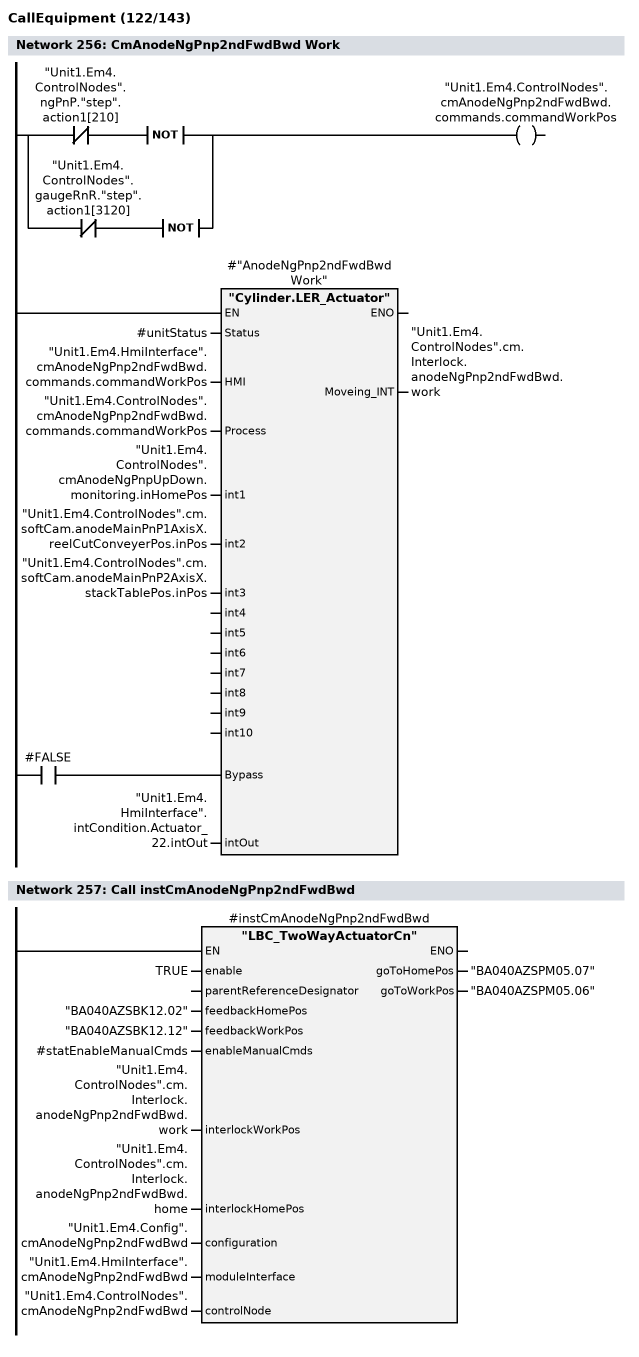
   RUNG wire#powerrail
      I_Contact( "Unit1.Em4.ControlNodes".ngPnP."step".action1[210] )
      Not()
      wire#w1
      Coil( "Unit1.Em4.ControlNodes".cmAnodeNgPnp2ndFwdBwd.commands.commandWorkPos )
   END_RUNG
   RUNG wire#powerrail
      I_Contact( "Unit1.Em4.ControlNodes".gaugeRnR."step".action1[3120] )
      Not()
   END_RUNG wire#w1
   RUNG wire#powerrail
      #"AnodeNgPnp2ndFwdBwd Work"(Bypass := wire#w2, Status := #unitStatus, HMI := "Unit1.Em4.HmiInterface".cmAnodeNgPnp2ndFwdBwd.commands.commandWorkPos, Process := "Unit1.Em4.ControlNodes".cmAnodeNgPnp2ndFwdBwd.commands.commandWorkPos, int1 := "Unit1.Em4.ControlNodes".cmAnodeNgPnpUpDown.monitoring.inHomePos, int2 := "Unit1.Em4.ControlNodes".cm.softCam.anodeMainPnP1AxisX.reelCutConveyerPos.inPos, int3 := "Unit1.Em4.ControlNodes".cm.softCam.anodeMainPnP2AxisX.stackTablePos.inPos, int4 :=, int5 :=, int6 :=, int7 :=, int8 :=, int9 :=, int10 :=, intOut := "Unit1.Em4.HmiInterface".intCondition.Actuator_22.intOut, Moveing_INT => "Unit1.Em4.ControlNodes".cm.Interlock.anodeNgPnp2ndFwdBwd.work)
   END_RUNG
   RUNG wire#powerrail
      Contact( #FALSE )
   END_RUNG wire#w2
   // the same network as SCL:
   "Unit1.Em4.ControlNodes".cmAnodeNgPnp2ndFwdBwd.commands.commandWorkPos := NOT (NOT "Unit1.Em4.ControlNodes".ngPnP."step".action1[210]) OR NOT (NOT "Unit1.Em4.ControlNodes".gaugeRnR."step".action1[3120]);
   #"AnodeNgPnp2ndFwdBwd Work"(Status := #unitStatus,   // "Cylinder.LER_Actuator"
                           HMI := "Unit1.Em4.HmiInterface".cmAnodeNgPnp2ndFwdBwd.commands.commandWorkPos,
                           Process := "Unit1.Em4.ControlNodes".cmAnodeNgPnp2ndFwdBwd.commands.commandWorkPos,
                           int1 := "Unit1.Em4.ControlNodes".cmAnodeNgPnpUpDown.monitoring.inHomePos,
                           int2 := "Unit1.Em4.ControlNodes".cm.softCam.anodeMainPnP1AxisX.reelCutConveyerPos.inPos,
                           int3 := "Unit1.Em4.ControlNodes".cm.softCam.anodeMainPnP2AxisX.stackTablePos.inPos,
                           Bypass := #FALSE,
                           intOut := "Unit1.Em4.HmiInterface".intCondition.Actuator_22.intOut,
                           Moveing_INT => "Unit1.Em4.ControlNodes".cm.Interlock.anodeNgPnp2ndFwdBwd.work);
END_REGION

REGION Network 257: Call instCmAnodeNgPnp2ndFwdBwd
   RUNG wire#powerrail
      #instCmAnodeNgPnp2ndFwdBwd(enable := TRUE, parentReferenceDesignator :=, feedbackHomePos := "BA040AZSBK12.02", feedbackWorkPos := "BA040AZSBK12.12", enableManualCmds := #statEnableManualCmds, interlockWorkPos := "Unit1.Em4.ControlNodes".cm.Interlock.anodeNgPnp2ndFwdBwd.work, interlockHomePos := "Unit1.Em4.ControlNodes".cm.Interlock.anodeNgPnp2ndFwdBwd.home, configuration := "Unit1.Em4.Config".cmAnodeNgPnp2ndFwdBwd, moduleInterface := "Unit1.Em4.HmiInterface".cmAnodeNgPnp2ndFwdBwd, controlNode := "Unit1.Em4.ControlNodes".cmAnodeNgPnp2ndFwdBwd, goToHomePos => "BA040AZSPM05.07", goToWorkPos => "BA040AZSPM05.06")
   END_RUNG
   // the same network as SCL:
   #instCmAnodeNgPnp2ndFwdBwd(enable := TRUE,   // "LBC_TwoWayActuatorCn"
                           feedbackHomePos := "BA040AZSBK12.02",
                           feedbackWorkPos := "BA040AZSBK12.12",
                           enableManualCmds := #statEnableManualCmds,
                           interlockWorkPos := "Unit1.Em4.ControlNodes".cm.Interlock.anodeNgPnp2ndFwdBwd.work,
                           interlockHomePos := "Unit1.Em4.ControlNodes".cm.Interlock.anodeNgPnp2ndFwdBwd.home,
                           configuration := "Unit1.Em4.Config".cmAnodeNgPnp2ndFwdBwd,
                           moduleInterface := "Unit1.Em4.HmiInterface".cmAnodeNgPnp2ndFwdBwd,
                           controlNode := "Unit1.Em4.ControlNodes".cmAnodeNgPnp2ndFwdBwd,
                           goToHomePos => "BA040AZSPM05.07",
                           goToWorkPos => "BA040AZSPM05.06");
END_REGION

REGION Network 259: CmAnodeMaintenanceMovingFixFrontRearFwdBwd Home
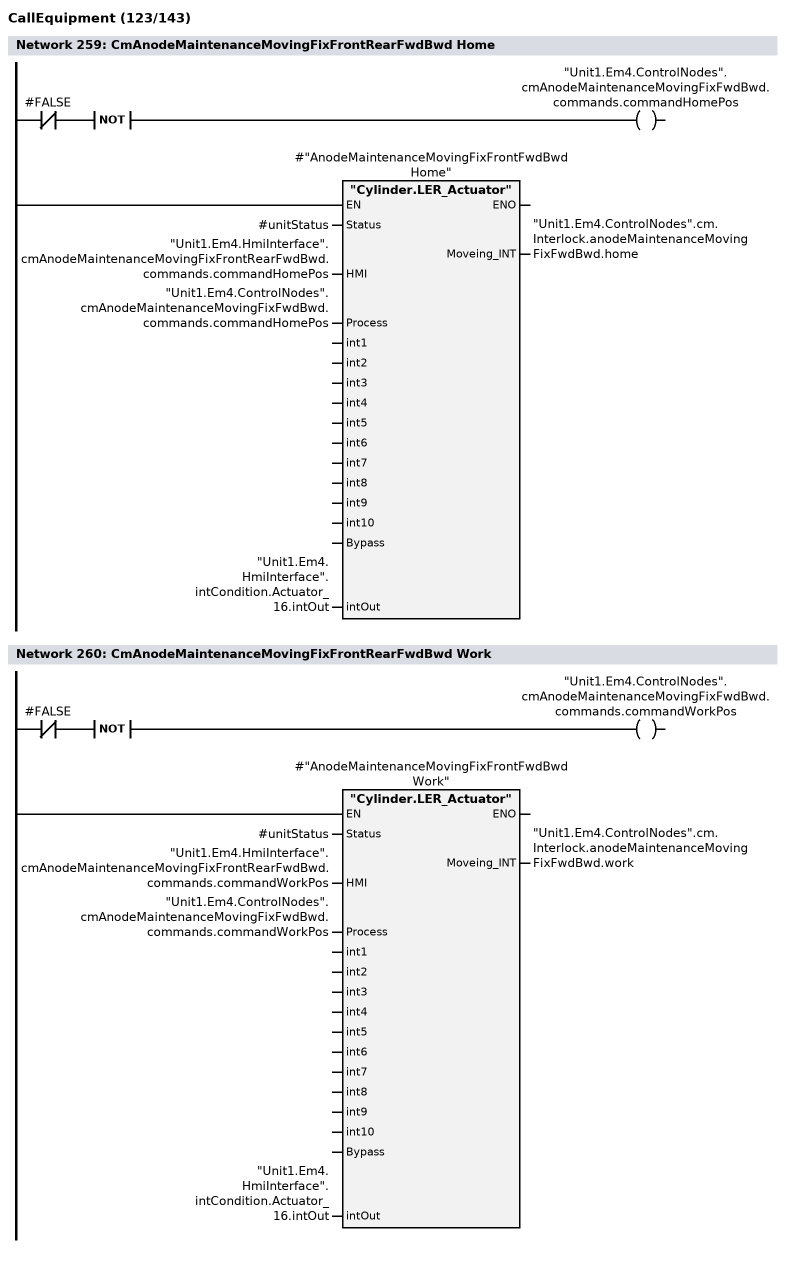
   RUNG wire#powerrail
      I_Contact( #FALSE )
      Not()
      Coil( "Unit1.Em4.ControlNodes".cmAnodeMaintenanceMovingFixFwdBwd.commands.commandHomePos )
   END_RUNG
   RUNG wire#powerrail
      #"AnodeMaintenanceMovingFixFrontFwdBwd Home"(Status := #unitStatus, HMI := "Unit1.Em4.HmiInterface".cmAnodeMaintenanceMovingFixFrontRearFwdBwd.commands.commandHomePos, Process := "Unit1.Em4.ControlNodes".cmAnodeMaintenanceMovingFixFwdBwd.commands.commandHomePos, int1 :=, int2 :=, int3 :=, int4 :=, int5 :=, int6 :=, int7 :=, int8 :=, int9 :=, int10 :=, Bypass :=, intOut := "Unit1.Em4.HmiInterface".intCondition.Actuator_16.intOut, Moveing_INT => "Unit1.Em4.ControlNodes".cm.Interlock.anodeMaintenanceMovingFixFwdBwd.home)
   END_RUNG
   // the same network as SCL:
   "Unit1.Em4.ControlNodes".cmAnodeMaintenanceMovingFixFwdBwd.commands.commandHomePos := NOT (NOT #FALSE);
   #"AnodeMaintenanceMovingFixFrontFwdBwd Home"(Status := #unitStatus,   // "Cylinder.LER_Actuator"
                           HMI := "Unit1.Em4.HmiInterface".cmAnodeMaintenanceMovingFixFrontRearFwdBwd.commands.commandHomePos,
                           Process := "Unit1.Em4.ControlNodes".cmAnodeMaintenanceMovingFixFwdBwd.commands.commandHomePos,
                           intOut := "Unit1.Em4.HmiInterface".intCondition.Actuator_16.intOut,
                           Moveing_INT => "Unit1.Em4.ControlNodes".cm.Interlock.anodeMaintenanceMovingFixFwdBwd.home);
END_REGION

REGION Network 260: CmAnodeMaintenanceMovingFixFrontRearFwdBwd Work
   RUNG wire#powerrail
      I_Contact( #FALSE )
      Not()
      Coil( "Unit1.Em4.ControlNodes".cmAnodeMaintenanceMovingFixFwdBwd.commands.commandWorkPos )
   END_RUNG
   RUNG wire#powerrail
      #"AnodeMaintenanceMovingFixFrontFwdBwd Work"(Status := #unitStatus, HMI := "Unit1.Em4.HmiInterface".cmAnodeMaintenanceMovingFixFrontRearFwdBwd.commands.commandWorkPos, Process := "Unit1.Em4.ControlNodes".cmAnodeMaintenanceMovingFixFwdBwd.commands.commandWorkPos, int1 :=, int2 :=, int3 :=, int4 :=, int5 :=, int6 :=, int7 :=, int8 :=, int9 :=, int10 :=, Bypass :=, intOut := "Unit1.Em4.HmiInterface".intCondition.Actuator_16.intOut, Moveing_INT => "Unit1.Em4.ControlNodes".cm.Interlock.anodeMaintenanceMovingFixFwdBwd.work)
   END_RUNG
   // the same network as SCL:
   "Unit1.Em4.ControlNodes".cmAnodeMaintenanceMovingFixFwdBwd.commands.commandWorkPos := NOT (NOT #FALSE);
   #"AnodeMaintenanceMovingFixFrontFwdBwd Work"(Status := #unitStatus,   // "Cylinder.LER_Actuator"
                           HMI := "Unit1.Em4.HmiInterface".cmAnodeMaintenanceMovingFixFrontRearFwdBwd.commands.commandWorkPos,
                           Process := "Unit1.Em4.ControlNodes".cmAnodeMaintenanceMovingFixFwdBwd.commands.commandWorkPos,
                           intOut := "Unit1.Em4.HmiInterface".intCondition.Actuator_16.intOut,
                           Moveing_INT => "Unit1.Em4.ControlNodes".cm.Interlock.anodeMaintenanceMovingFixFwdBwd.work);
END_REGION

REGION Network 261: Call instCmAnodeMaintenanceMovingFixFrontRearFwdBwd
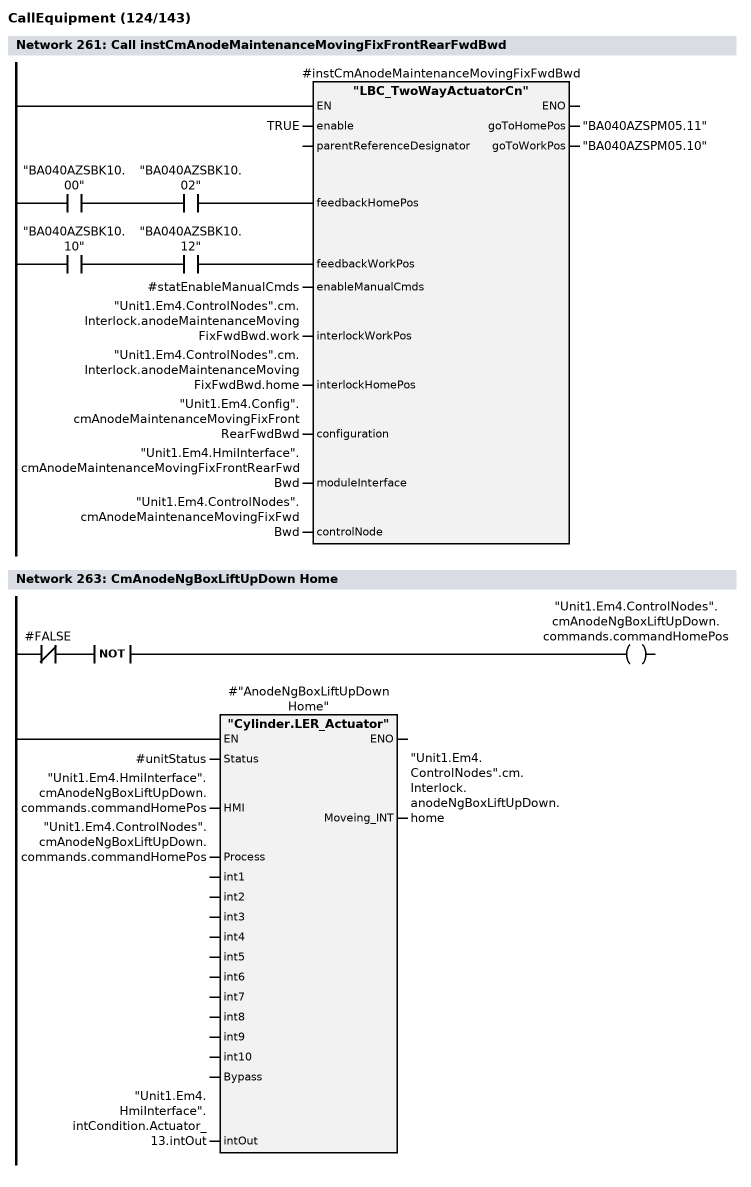
   RUNG wire#powerrail
      #instCmAnodeMaintenanceMovingFixFwdBwd(feedbackHomePos := wire#w1, feedbackWorkPos := wire#w2, enable := TRUE, parentReferenceDesignator :=, enableManualCmds := #statEnableManualCmds, interlockWorkPos := "Unit1.Em4.ControlNodes".cm.Interlock.anodeMaintenanceMovingFixFwdBwd.work, interlockHomePos := "Unit1.Em4.ControlNodes".cm.Interlock.anodeMaintenanceMovingFixFwdBwd.home, configuration := "Unit1.Em4.Config".cmAnodeMaintenanceMovingFixFrontRearFwdBwd, moduleInterface := "Unit1.Em4.HmiInterface".cmAnodeMaintenanceMovingFixFrontRearFwdBwd, controlNode := "Unit1.Em4.ControlNodes".cmAnodeMaintenanceMovingFixFwdBwd, goToHomePos => "BA040AZSPM05.11", goToWorkPos => "BA040AZSPM05.10")
   END_RUNG
   RUNG wire#powerrail
      Contact( "BA040AZSBK10.00" )
      Contact( "BA040AZSBK10.02" )
   END_RUNG wire#w1
   RUNG wire#powerrail
      Contact( "BA040AZSBK10.10" )
      Contact( "BA040AZSBK10.12" )
   END_RUNG wire#w2
   // the same network as SCL:
   #instCmAnodeMaintenanceMovingFixFwdBwd(enable := TRUE,   // "LBC_TwoWayActuatorCn"
                           feedbackHomePos := "BA040AZSBK10.00" AND "BA040AZSBK10.02",
                           feedbackWorkPos := "BA040AZSBK10.10" AND "BA040AZSBK10.12",
                           enableManualCmds := #statEnableManualCmds,
                           interlockWorkPos := "Unit1.Em4.ControlNodes".cm.Interlock.anodeMaintenanceMovingFixFwdBwd.work,
                           interlockHomePos := "Unit1.Em4.ControlNodes".cm.Interlock.anodeMaintenanceMovingFixFwdBwd.home,
                           configuration := "Unit1.Em4.Config".cmAnodeMaintenanceMovingFixFrontRearFwdBwd,
                           moduleInterface := "Unit1.Em4.HmiInterface".cmAnodeMaintenanceMovingFixFrontRearFwdBwd,
                           controlNode := "Unit1.Em4.ControlNodes".cmAnodeMaintenanceMovingFixFwdBwd,
                           goToHomePos => "BA040AZSPM05.11",
                           goToWorkPos => "BA040AZSPM05.10");
END_REGION

REGION Network 263: CmAnodeNgBoxLiftUpDown Home
   RUNG wire#powerrail
      I_Contact( #FALSE )
      Not()
      Coil( "Unit1.Em4.ControlNodes".cmAnodeNgBoxLiftUpDown.commands.commandHomePos )
   END_RUNG
   RUNG wire#powerrail
      #"AnodeNgBoxLiftUpDown Home"(Status := #unitStatus, HMI := "Unit1.Em4.HmiInterface".cmAnodeNgBoxLiftUpDown.commands.commandHomePos, Process := "Unit1.Em4.ControlNodes".cmAnodeNgBoxLiftUpDown.commands.commandHomePos, int1 :=, int2 :=, int3 :=, int4 :=, int5 :=, int6 :=, int7 :=, int8 :=, int9 :=, int10 :=, Bypass :=, intOut := "Unit1.Em4.HmiInterface".intCondition.Actuator_13.intOut, Moveing_INT => "Unit1.Em4.ControlNodes".cm.Interlock.anodeNgBoxLiftUpDown.home)
   END_RUNG
   // the same network as SCL:
   "Unit1.Em4.ControlNodes".cmAnodeNgBoxLiftUpDown.commands.commandHomePos := NOT (NOT #FALSE);
   #"AnodeNgBoxLiftUpDown Home"(Status := #unitStatus,   // "Cylinder.LER_Actuator"
                           HMI := "Unit1.Em4.HmiInterface".cmAnodeNgBoxLiftUpDown.commands.commandHomePos,
                           Process := "Unit1.Em4.ControlNodes".cmAnodeNgBoxLiftUpDown.commands.commandHomePos,
                           intOut := "Unit1.Em4.HmiInterface".intCondition.Actuator_13.intOut,
                           Moveing_INT => "Unit1.Em4.ControlNodes".cm.Interlock.anodeNgBoxLiftUpDown.home);
END_REGION

REGION Network 264: CmAnodeNgBoxLiftUpDown Work
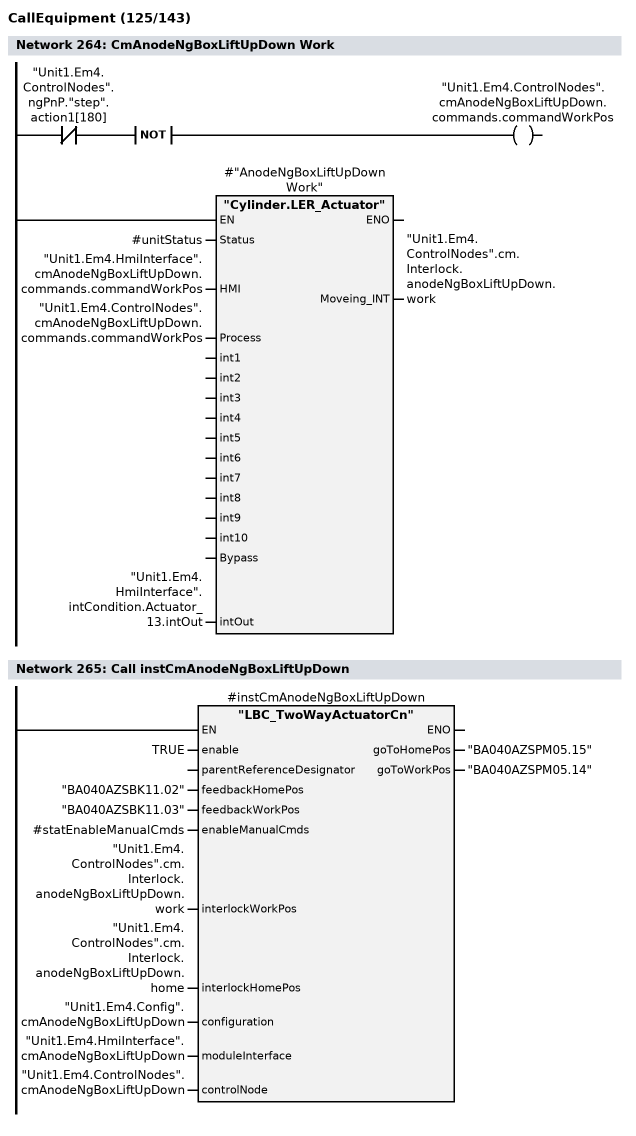
   RUNG wire#powerrail
      I_Contact( "Unit1.Em4.ControlNodes".ngPnP."step".action1[180] )
      Not()
      Coil( "Unit1.Em4.ControlNodes".cmAnodeNgBoxLiftUpDown.commands.commandWorkPos )
   END_RUNG
   RUNG wire#powerrail
      #"AnodeNgBoxLiftUpDown Work"(Status := #unitStatus, HMI := "Unit1.Em4.HmiInterface".cmAnodeNgBoxLiftUpDown.commands.commandWorkPos, Process := "Unit1.Em4.ControlNodes".cmAnodeNgBoxLiftUpDown.commands.commandWorkPos, int1 :=, int2 :=, int3 :=, int4 :=, int5 :=, int6 :=, int7 :=, int8 :=, int9 :=, int10 :=, Bypass :=, intOut := "Unit1.Em4.HmiInterface".intCondition.Actuator_13.intOut, Moveing_INT => "Unit1.Em4.ControlNodes".cm.Interlock.anodeNgBoxLiftUpDown.work)
   END_RUNG
   // the same network as SCL:
   "Unit1.Em4.ControlNodes".cmAnodeNgBoxLiftUpDown.commands.commandWorkPos := NOT (NOT "Unit1.Em4.ControlNodes".ngPnP."step".action1[180]);
   #"AnodeNgBoxLiftUpDown Work"(Status := #unitStatus,   // "Cylinder.LER_Actuator"
                           HMI := "Unit1.Em4.HmiInterface".cmAnodeNgBoxLiftUpDown.commands.commandWorkPos,
                           Process := "Unit1.Em4.ControlNodes".cmAnodeNgBoxLiftUpDown.commands.commandWorkPos,
                           intOut := "Unit1.Em4.HmiInterface".intCondition.Actuator_13.intOut,
                           Moveing_INT => "Unit1.Em4.ControlNodes".cm.Interlock.anodeNgBoxLiftUpDown.work);
END_REGION

REGION Network 265: Call instCmAnodeNgBoxLiftUpDown
   RUNG wire#powerrail
      #instCmAnodeNgBoxLiftUpDown(enable := TRUE, parentReferenceDesignator :=, feedbackHomePos := "BA040AZSBK11.02", feedbackWorkPos := "BA040AZSBK11.03", enableManualCmds := #statEnableManualCmds, interlockWorkPos := "Unit1.Em4.ControlNodes".cm.Interlock.anodeNgBoxLiftUpDown.work, interlockHomePos := "Unit1.Em4.ControlNodes".cm.Interlock.anodeNgBoxLiftUpDown.home, configuration := "Unit1.Em4.Config".cmAnodeNgBoxLiftUpDown, moduleInterface := "Unit1.Em4.HmiInterface".cmAnodeNgBoxLiftUpDown, controlNode := "Unit1.Em4.ControlNodes".cmAnodeNgBoxLiftUpDown, goToHomePos => "BA040AZSPM05.15", goToWorkPos => "BA040AZSPM05.14")
   END_RUNG
   // the same network as SCL:
   #instCmAnodeNgBoxLiftUpDown(enable := TRUE,   // "LBC_TwoWayActuatorCn"
                           feedbackHomePos := "BA040AZSBK11.02",
                           feedbackWorkPos := "BA040AZSBK11.03",
                           enableManualCmds := #statEnableManualCmds,
                           interlockWorkPos := "Unit1.Em4.ControlNodes".cm.Interlock.anodeNgBoxLiftUpDown.work,
                           interlockHomePos := "Unit1.Em4.ControlNodes".cm.Interlock.anodeNgBoxLiftUpDown.home,
                           configuration := "Unit1.Em4.Config".cmAnodeNgBoxLiftUpDown,
                           moduleInterface := "Unit1.Em4.HmiInterface".cmAnodeNgBoxLiftUpDown,
                           controlNode := "Unit1.Em4.ControlNodes".cmAnodeNgBoxLiftUpDown,
                           goToHomePos => "BA040AZSPM05.15",
                           goToWorkPos => "BA040AZSPM05.14");
END_REGION

REGION Network 267: CmAnodeNgBoxLockUpDown Home
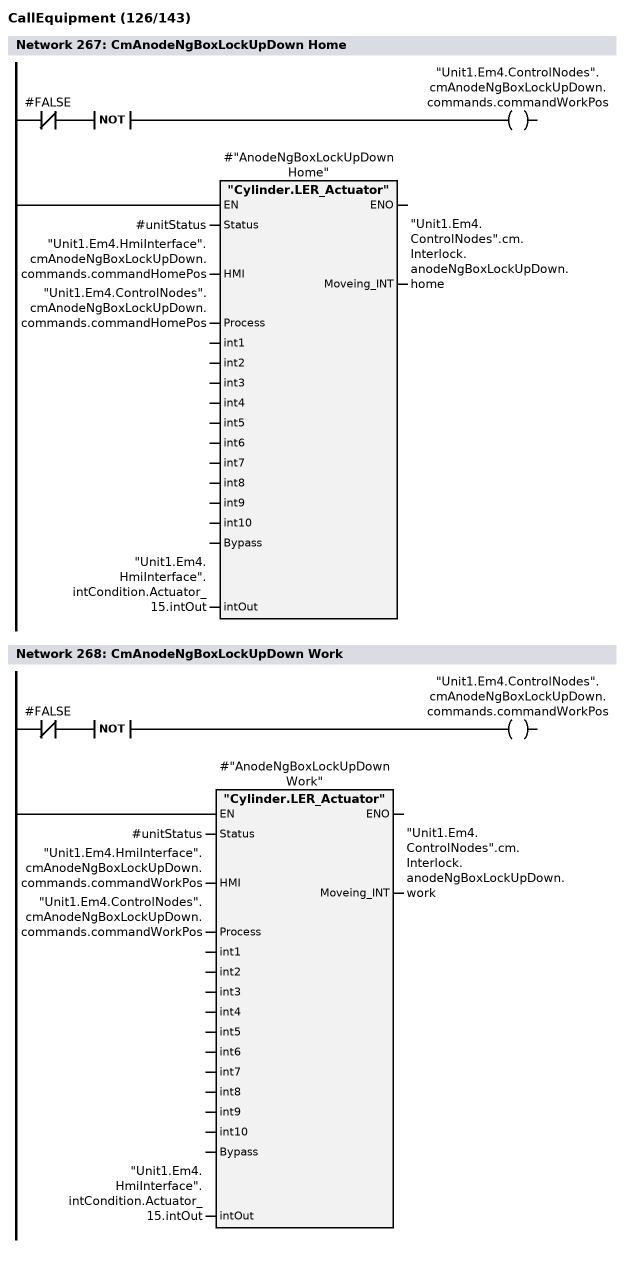
   RUNG wire#powerrail
      I_Contact( #FALSE )
      Not()
      Coil( "Unit1.Em4.ControlNodes".cmAnodeNgBoxLockUpDown.commands.commandWorkPos )
   END_RUNG
   RUNG wire#powerrail
      #"AnodeNgBoxLockUpDown Home"(Status := #unitStatus, HMI := "Unit1.Em4.HmiInterface".cmAnodeNgBoxLockUpDown.commands.commandHomePos, Process := "Unit1.Em4.ControlNodes".cmAnodeNgBoxLockUpDown.commands.commandHomePos, int1 :=, int2 :=, int3 :=, int4 :=, int5 :=, int6 :=, int7 :=, int8 :=, int9 :=, int10 :=, Bypass :=, intOut := "Unit1.Em4.HmiInterface".intCondition.Actuator_15.intOut, Moveing_INT => "Unit1.Em4.ControlNodes".cm.Interlock.anodeNgBoxLockUpDown.home)
   END_RUNG
   // the same network as SCL:
   "Unit1.Em4.ControlNodes".cmAnodeNgBoxLockUpDown.commands.commandWorkPos := NOT (NOT #FALSE);
   #"AnodeNgBoxLockUpDown Home"(Status := #unitStatus,   // "Cylinder.LER_Actuator"
                           HMI := "Unit1.Em4.HmiInterface".cmAnodeNgBoxLockUpDown.commands.commandHomePos,
                           Process := "Unit1.Em4.ControlNodes".cmAnodeNgBoxLockUpDown.commands.commandHomePos,
                           intOut := "Unit1.Em4.HmiInterface".intCondition.Actuator_15.intOut,
                           Moveing_INT => "Unit1.Em4.ControlNodes".cm.Interlock.anodeNgBoxLockUpDown.home);
END_REGION

REGION Network 268: CmAnodeNgBoxLockUpDown Work
   RUNG wire#powerrail
      I_Contact( #FALSE )
      Not()
      Coil( "Unit1.Em4.ControlNodes".cmAnodeNgBoxLockUpDown.commands.commandWorkPos )
   END_RUNG
   RUNG wire#powerrail
      #"AnodeNgBoxLockUpDown Work"(Status := #unitStatus, HMI := "Unit1.Em4.HmiInterface".cmAnodeNgBoxLockUpDown.commands.commandWorkPos, Process := "Unit1.Em4.ControlNodes".cmAnodeNgBoxLockUpDown.commands.commandWorkPos, int1 :=, int2 :=, int3 :=, int4 :=, int5 :=, int6 :=, int7 :=, int8 :=, int9 :=, int10 :=, Bypass :=, intOut := "Unit1.Em4.HmiInterface".intCondition.Actuator_15.intOut, Moveing_INT => "Unit1.Em4.ControlNodes".cm.Interlock.anodeNgBoxLockUpDown.work)
   END_RUNG
   // the same network as SCL:
   "Unit1.Em4.ControlNodes".cmAnodeNgBoxLockUpDown.commands.commandWorkPos := NOT (NOT #FALSE);
   #"AnodeNgBoxLockUpDown Work"(Status := #unitStatus,   // "Cylinder.LER_Actuator"
                           HMI := "Unit1.Em4.HmiInterface".cmAnodeNgBoxLockUpDown.commands.commandWorkPos,
                           Process := "Unit1.Em4.ControlNodes".cmAnodeNgBoxLockUpDown.commands.commandWorkPos,
                           intOut := "Unit1.Em4.HmiInterface".intCondition.Actuator_15.intOut,
                           Moveing_INT => "Unit1.Em4.ControlNodes".cm.Interlock.anodeNgBoxLockUpDown.work);
END_REGION

REGION Network 269: Call instCmAnodeNgBoxLockUpDown
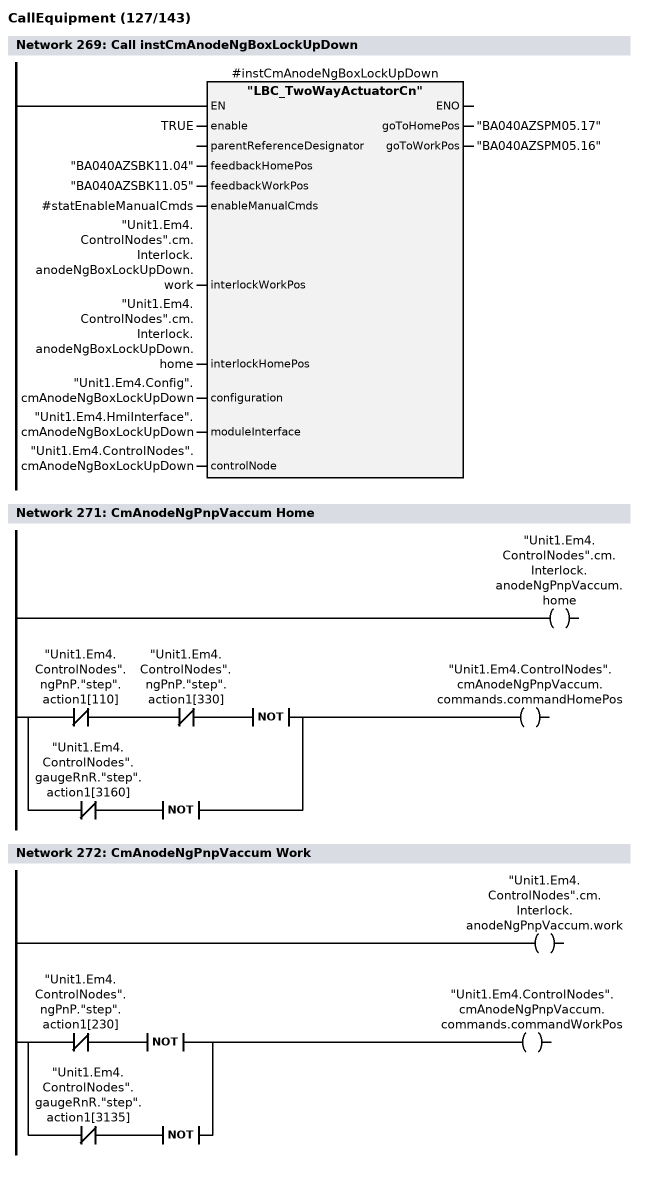
   RUNG wire#powerrail
      #instCmAnodeNgBoxLockUpDown(enable := TRUE, parentReferenceDesignator :=, feedbackHomePos := "BA040AZSBK11.04", feedbackWorkPos := "BA040AZSBK11.05", enableManualCmds := #statEnableManualCmds, interlockWorkPos := "Unit1.Em4.ControlNodes".cm.Interlock.anodeNgBoxLockUpDown.work, interlockHomePos := "Unit1.Em4.ControlNodes".cm.Interlock.anodeNgBoxLockUpDown.home, configuration := "Unit1.Em4.Config".cmAnodeNgBoxLockUpDown, moduleInterface := "Unit1.Em4.HmiInterface".cmAnodeNgBoxLockUpDown, controlNode := "Unit1.Em4.ControlNodes".cmAnodeNgBoxLockUpDown, goToHomePos => "BA040AZSPM05.17", goToWorkPos => "BA040AZSPM05.16")
   END_RUNG
   // the same network as SCL:
   #instCmAnodeNgBoxLockUpDown(enable := TRUE,   // "LBC_TwoWayActuatorCn"
                           feedbackHomePos := "BA040AZSBK11.04",
                           feedbackWorkPos := "BA040AZSBK11.05",
                           enableManualCmds := #statEnableManualCmds,
                           interlockWorkPos := "Unit1.Em4.ControlNodes".cm.Interlock.anodeNgBoxLockUpDown.work,
                           interlockHomePos := "Unit1.Em4.ControlNodes".cm.Interlock.anodeNgBoxLockUpDown.home,
                           configuration := "Unit1.Em4.Config".cmAnodeNgBoxLockUpDown,
                           moduleInterface := "Unit1.Em4.HmiInterface".cmAnodeNgBoxLockUpDown,
                           controlNode := "Unit1.Em4.ControlNodes".cmAnodeNgBoxLockUpDown,
                           goToHomePos => "BA040AZSPM05.17",
                           goToWorkPos => "BA040AZSPM05.16");
END_REGION

REGION Network 271: CmAnodeNgPnpVaccum Home
   RUNG wire#powerrail
      Coil( "Unit1.Em4.ControlNodes".cm.Interlock.anodeNgPnpVaccum.home )
   END_RUNG
   RUNG wire#powerrail
      I_Contact( "Unit1.Em4.ControlNodes".ngPnP."step".action1[110] )
      I_Contact( "Unit1.Em4.ControlNodes".ngPnP."step".action1[330] )
      Not()
      wire#w1
      Coil( "Unit1.Em4.ControlNodes".cmAnodeNgPnpVaccum.commands.commandHomePos )
   END_RUNG
   RUNG wire#powerrail
      I_Contact( "Unit1.Em4.ControlNodes".gaugeRnR."step".action1[3160] )
      Not()
   END_RUNG wire#w1
   // the same network as SCL:
   "Unit1.Em4.ControlNodes".cm.Interlock.anodeNgPnpVaccum.home := TRUE;
   "Unit1.Em4.ControlNodes".cmAnodeNgPnpVaccum.commands.commandHomePos := NOT (NOT "Unit1.Em4.ControlNodes".ngPnP."step".action1[110] AND NOT "Unit1.Em4.ControlNodes".ngPnP."step".action1[330]) OR NOT (NOT "Unit1.Em4.ControlNodes".gaugeRnR."step".action1[3160]);
END_REGION

REGION Network 272: CmAnodeNgPnpVaccum Work
   RUNG wire#powerrail
      Coil( "Unit1.Em4.ControlNodes".cm.Interlock.anodeNgPnpVaccum.work )
   END_RUNG
   RUNG wire#powerrail
      I_Contact( "Unit1.Em4.ControlNodes".ngPnP."step".action1[230] )
      Not()
      wire#w1
      Coil( "Unit1.Em4.ControlNodes".cmAnodeNgPnpVaccum.commands.commandWorkPos )
   END_RUNG
   RUNG wire#powerrail
      I_Contact( "Unit1.Em4.ControlNodes".gaugeRnR."step".action1[3135] )
      Not()
   END_RUNG wire#w1
   // the same network as SCL:
   "Unit1.Em4.ControlNodes".cm.Interlock.anodeNgPnpVaccum.work := TRUE;
   "Unit1.Em4.ControlNodes".cmAnodeNgPnpVaccum.commands.commandWorkPos := NOT (NOT "Unit1.Em4.ControlNodes".ngPnP."step".action1[230]) OR NOT (NOT "Unit1.Em4.ControlNodes".gaugeRnR."step".action1[3135]);
END_REGION

REGION Network 273: Call instCmAnodeNgPnpVaccum
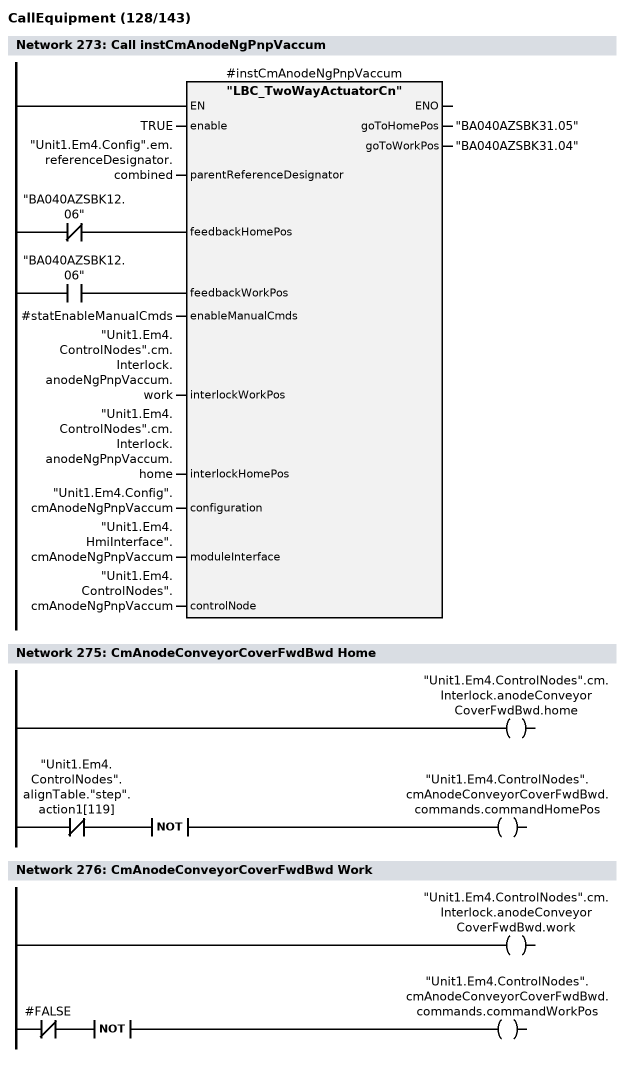
   RUNG wire#powerrail
      #instCmAnodeNgPnpVaccum(feedbackHomePos := wire#w1, feedbackWorkPos := wire#w2, enable := TRUE, parentReferenceDesignator := "Unit1.Em4.Config".em.referenceDesignator.combined, enableManualCmds := #statEnableManualCmds, interlockWorkPos := "Unit1.Em4.ControlNodes".cm.Interlock.anodeNgPnpVaccum.work, interlockHomePos := "Unit1.Em4.ControlNodes".cm.Interlock.anodeNgPnpVaccum.home, configuration := "Unit1.Em4.Config".cmAnodeNgPnpVaccum, moduleInterface := "Unit1.Em4.HmiInterface".cmAnodeNgPnpVaccum, controlNode := "Unit1.Em4.ControlNodes".cmAnodeNgPnpVaccum, goToHomePos => "BA040AZSBK31.05", goToWorkPos => "BA040AZSBK31.04")
   END_RUNG
   RUNG wire#powerrail
      I_Contact( "BA040AZSBK12.06" )
   END_RUNG wire#w1
   RUNG wire#powerrail
      Contact( "BA040AZSBK12.06" )
   END_RUNG wire#w2
   // the same network as SCL:
   #instCmAnodeNgPnpVaccum(enable := TRUE,   // "LBC_TwoWayActuatorCn"
                           parentReferenceDesignator := "Unit1.Em4.Config".em.referenceDesignator.combined,
                           feedbackHomePos := NOT "BA040AZSBK12.06",
                           feedbackWorkPos := "BA040AZSBK12.06",
                           enableManualCmds := #statEnableManualCmds,
                           interlockWorkPos := "Unit1.Em4.ControlNodes".cm.Interlock.anodeNgPnpVaccum.work,
                           interlockHomePos := "Unit1.Em4.ControlNodes".cm.Interlock.anodeNgPnpVaccum.home,
                           configuration := "Unit1.Em4.Config".cmAnodeNgPnpVaccum,
                           moduleInterface := "Unit1.Em4.HmiInterface".cmAnodeNgPnpVaccum,
                           controlNode := "Unit1.Em4.ControlNodes".cmAnodeNgPnpVaccum,
                           goToHomePos => "BA040AZSBK31.05",
                           goToWorkPos => "BA040AZSBK31.04");
END_REGION

REGION Network 275: CmAnodeConveyorCoverFwdBwd Home
   RUNG wire#powerrail
      Coil( "Unit1.Em4.ControlNodes".cm.Interlock.anodeConveyorCoverFwdBwd.home )
   END_RUNG
   RUNG wire#powerrail
      I_Contact( "Unit1.Em4.ControlNodes".alignTable."step".action1[119] )
      Not()
      Coil( "Unit1.Em4.ControlNodes".cmAnodeConveyorCoverFwdBwd.commands.commandHomePos )
   END_RUNG
   // the same network as SCL:
   "Unit1.Em4.ControlNodes".cm.Interlock.anodeConveyorCoverFwdBwd.home := TRUE;
   "Unit1.Em4.ControlNodes".cmAnodeConveyorCoverFwdBwd.commands.commandHomePos := NOT (NOT "Unit1.Em4.ControlNodes".alignTable."step".action1[119]);
END_REGION

REGION Network 276: CmAnodeConveyorCoverFwdBwd Work
   RUNG wire#powerrail
      Coil( "Unit1.Em4.ControlNodes".cm.Interlock.anodeConveyorCoverFwdBwd.work )
   END_RUNG
   RUNG wire#powerrail
      I_Contact( #FALSE )
      Not()
      Coil( "Unit1.Em4.ControlNodes".cmAnodeConveyorCoverFwdBwd.commands.commandWorkPos )
   END_RUNG
   // the same network as SCL:
   "Unit1.Em4.ControlNodes".cm.Interlock.anodeConveyorCoverFwdBwd.work := TRUE;
   "Unit1.Em4.ControlNodes".cmAnodeConveyorCoverFwdBwd.commands.commandWorkPos := NOT (NOT #FALSE);
END_REGION

REGION Network 277: Call instCmAnodeConveyorCoverFwdBwd
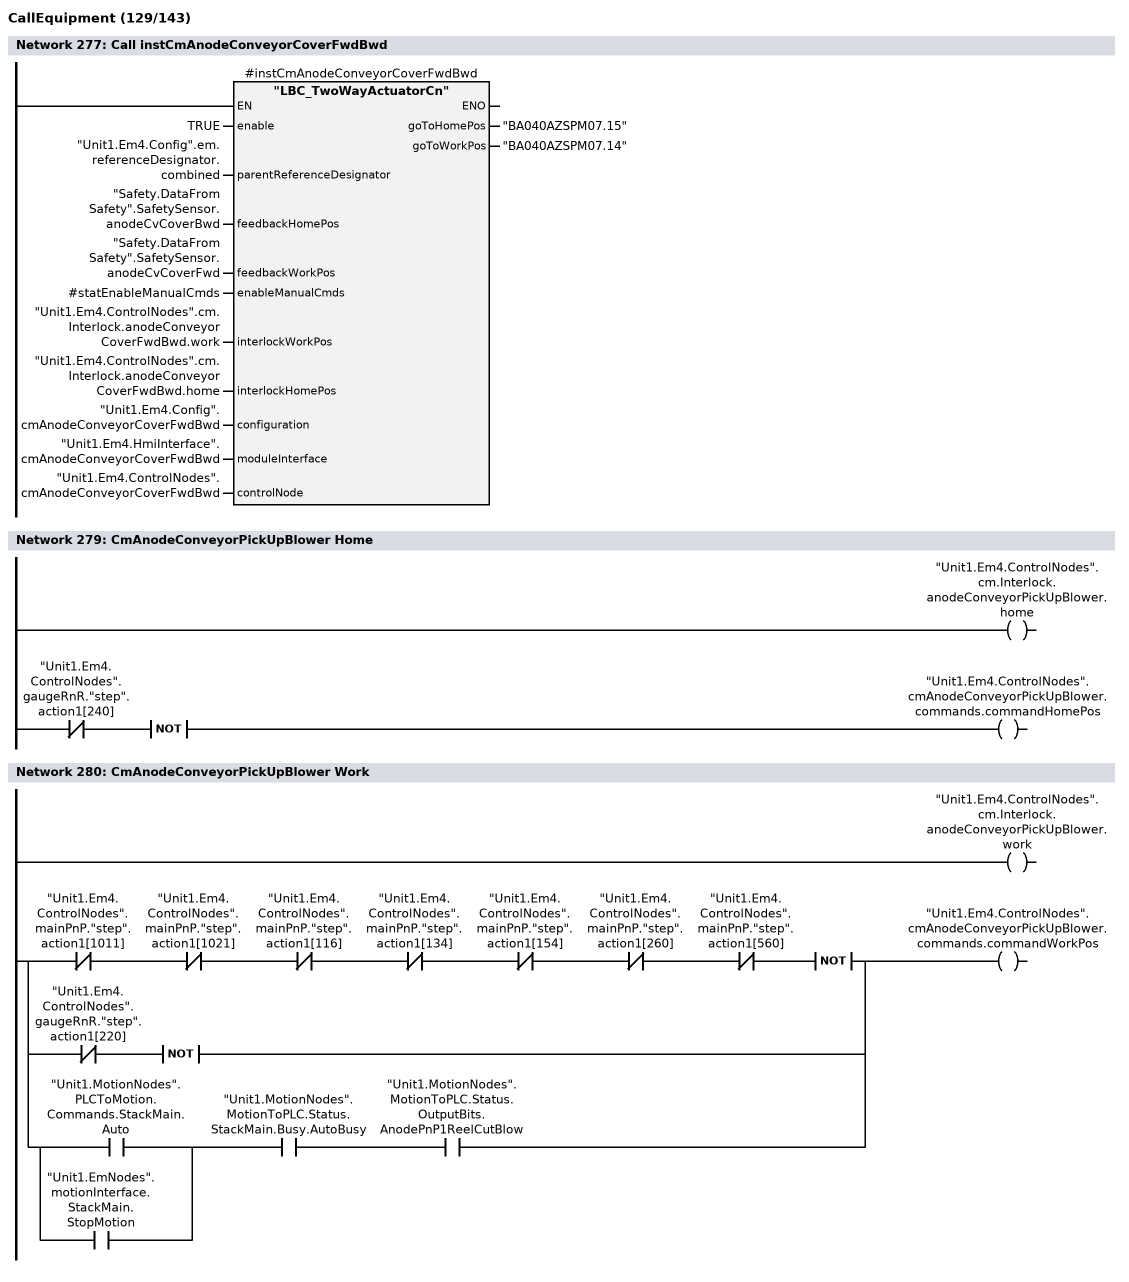
   RUNG wire#powerrail
      #instCmAnodeConveyorCoverFwdBwd(enable := TRUE, parentReferenceDesignator := "Unit1.Em4.Config".em.referenceDesignator.combined, feedbackHomePos := "Safety.DataFromSafety".SafetySensor.anodeCvCoverBwd, feedbackWorkPos := "Safety.DataFromSafety".SafetySensor.anodeCvCoverFwd, enableManualCmds := #statEnableManualCmds, interlockWorkPos := "Unit1.Em4.ControlNodes".cm.Interlock.anodeConveyorCoverFwdBwd.work, interlockHomePos := "Unit1.Em4.ControlNodes".cm.Interlock.anodeConveyorCoverFwdBwd.home, configuration := "Unit1.Em4.Config".cmAnodeConveyorCoverFwdBwd, moduleInterface := "Unit1.Em4.HmiInterface".cmAnodeConveyorCoverFwdBwd, controlNode := "Unit1.Em4.ControlNodes".cmAnodeConveyorCoverFwdBwd, goToHomePos => "BA040AZSPM07.15", goToWorkPos => "BA040AZSPM07.14")
   END_RUNG
   // the same network as SCL:
   #instCmAnodeConveyorCoverFwdBwd(enable := TRUE,   // "LBC_TwoWayActuatorCn"
                           parentReferenceDesignator := "Unit1.Em4.Config".em.referenceDesignator.combined,
                           feedbackHomePos := "Safety.DataFromSafety".SafetySensor.anodeCvCoverBwd,
                           feedbackWorkPos := "Safety.DataFromSafety".SafetySensor.anodeCvCoverFwd,
                           enableManualCmds := #statEnableManualCmds,
                           interlockWorkPos := "Unit1.Em4.ControlNodes".cm.Interlock.anodeConveyorCoverFwdBwd.work,
                           interlockHomePos := "Unit1.Em4.ControlNodes".cm.Interlock.anodeConveyorCoverFwdBwd.home,
                           configuration := "Unit1.Em4.Config".cmAnodeConveyorCoverFwdBwd,
                           moduleInterface := "Unit1.Em4.HmiInterface".cmAnodeConveyorCoverFwdBwd,
                           controlNode := "Unit1.Em4.ControlNodes".cmAnodeConveyorCoverFwdBwd,
                           goToHomePos => "BA040AZSPM07.15",
                           goToWorkPos => "BA040AZSPM07.14");
END_REGION

REGION Network 279: CmAnodeConveyorPickUpBlower Home
   RUNG wire#powerrail
      Coil( "Unit1.Em4.ControlNodes".cm.Interlock.anodeConveyorPickUpBlower.home )
   END_RUNG
   RUNG wire#powerrail
      I_Contact( "Unit1.Em4.ControlNodes".gaugeRnR."step".action1[240] )
      Not()
      Coil( "Unit1.Em4.ControlNodes".cmAnodeConveyorPickUpBlower.commands.commandHomePos )
   END_RUNG
   // the same network as SCL:
   "Unit1.Em4.ControlNodes".cm.Interlock.anodeConveyorPickUpBlower.home := TRUE;
   "Unit1.Em4.ControlNodes".cmAnodeConveyorPickUpBlower.commands.commandHomePos := NOT (NOT "Unit1.Em4.ControlNodes".gaugeRnR."step".action1[240]);
END_REGION

REGION Network 280: CmAnodeConveyorPickUpBlower Work
   RUNG wire#powerrail
      Coil( "Unit1.Em4.ControlNodes".cm.Interlock.anodeConveyorPickUpBlower.work )
   END_RUNG
   RUNG wire#powerrail
      I_Contact( "Unit1.Em4.ControlNodes".mainPnP."step".action1[1011] )
      I_Contact( "Unit1.Em4.ControlNodes".mainPnP."step".action1[1021] )
      I_Contact( "Unit1.Em4.ControlNodes".mainPnP."step".action1[116] )
      I_Contact( "Unit1.Em4.ControlNodes".mainPnP."step".action1[134] )
      I_Contact( "Unit1.Em4.ControlNodes".mainPnP."step".action1[154] )
      I_Contact( "Unit1.Em4.ControlNodes".mainPnP."step".action1[260] )
      I_Contact( "Unit1.Em4.ControlNodes".mainPnP."step".action1[560] )
      Not()
      wire#w1
      Coil( "Unit1.Em4.ControlNodes".cmAnodeConveyorPickUpBlower.commands.commandWorkPos )
   END_RUNG
   RUNG wire#powerrail
      I_Contact( "Unit1.Em4.ControlNodes".gaugeRnR."step".action1[220] )
      Not()
   END_RUNG wire#w1
   RUNG wire#powerrail
      Contact( "Unit1.MotionNodes".PLCToMotion.Commands.StackMain.Auto )
      wire#w2
      Contact( "Unit1.MotionNodes".MotionToPLC.Status.StackMain.Busy.AutoBusy )
      Contact( "Unit1.MotionNodes".MotionToPLC.Status.OutputBits.AnodePnP1ReelCutBlow )
   END_RUNG wire#w1
   RUNG wire#powerrail
      Contact( "Unit1.EmNodes".motionInterface.StackMain.StopMotion )
   END_RUNG wire#w2
   // the same network as SCL:
   "Unit1.Em4.ControlNodes".cm.Interlock.anodeConveyorPickUpBlower.work := TRUE;
   "Unit1.Em4.ControlNodes".cmAnodeConveyorPickUpBlower.commands.commandWorkPos := NOT (NOT "Unit1.Em4.ControlNodes".mainPnP."step".action1[1011] AND NOT "Unit1.Em4.ControlNodes".mainPnP."step".action1[1021] AND NOT "Unit1.Em4.ControlNodes".mainPnP."step".action1[116] AND NOT "Unit1.Em4.ControlNodes".mainPnP."step".action1[134] AND NOT "Unit1.Em4.ControlNodes".mainPnP."step".action1[154] AND NOT "Unit1.Em4.ControlNodes".mainPnP."step".action1[260] AND NOT "Unit1.Em4.ControlNodes".mainPnP."step".action1[560]) OR NOT (NOT "Unit1.Em4.ControlNodes".gaugeRnR."step".action1[220]) OR (("Unit1.MotionNodes".PLCToMotion.Commands.StackMain.Auto OR "Unit1.EmNodes".motionInterface.StackMain.StopMotion) AND "Unit1.MotionNodes".MotionToPLC.Status.StackMain.Busy.AutoBusy AND "Unit1.MotionNodes".MotionToPLC.Status.OutputBits.AnodePnP1ReelCutBlow);
END_REGION

REGION Network 281: Call instCmAnodeConveyorPickUpBlower
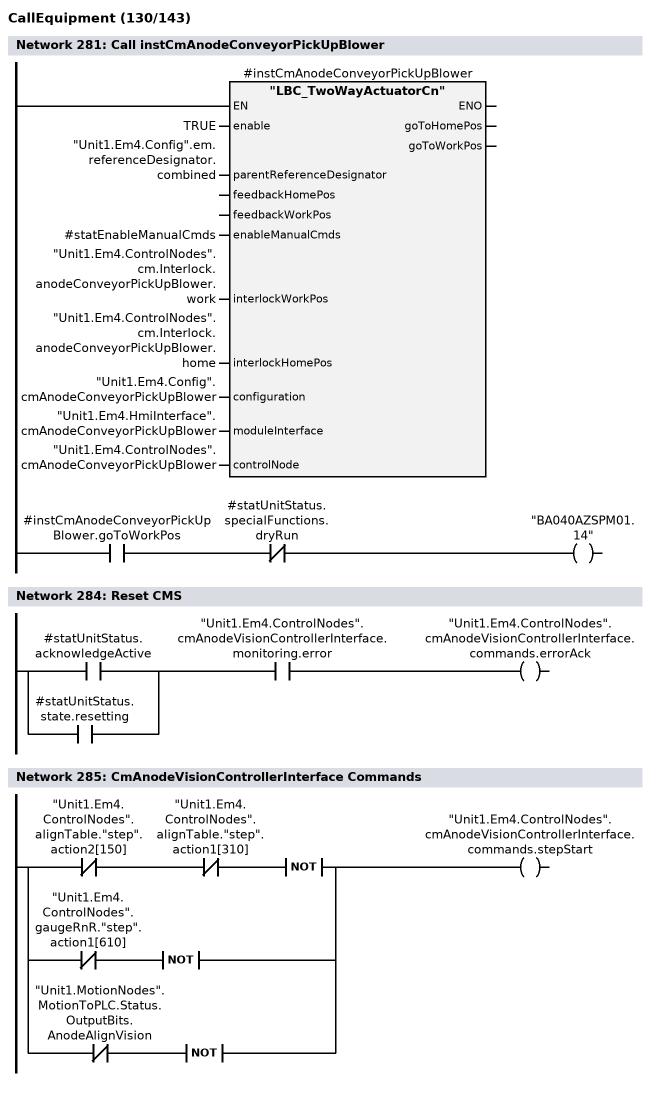
   RUNG wire#powerrail
      #instCmAnodeConveyorPickUpBlower(enable := TRUE, parentReferenceDesignator := "Unit1.Em4.Config".em.referenceDesignator.combined, feedbackHomePos :=, feedbackWorkPos :=, enableManualCmds := #statEnableManualCmds, interlockWorkPos := "Unit1.Em4.ControlNodes".cm.Interlock.anodeConveyorPickUpBlower.work, interlockHomePos := "Unit1.Em4.ControlNodes".cm.Interlock.anodeConveyorPickUpBlower.home, configuration := "Unit1.Em4.Config".cmAnodeConveyorPickUpBlower, moduleInterface := "Unit1.Em4.HmiInterface".cmAnodeConveyorPickUpBlower, controlNode := "Unit1.Em4.ControlNodes".cmAnodeConveyorPickUpBlower, goToHomePos =>, goToWorkPos =>)
   END_RUNG
   RUNG wire#powerrail
      Contact( #instCmAnodeConveyorPickUpBlower.goToWorkPos )
      I_Contact( #statUnitStatus.specialFunctions.dryRun )
      Coil( "BA040AZSPM01.14" )
   END_RUNG
   // the same network as SCL:
   #instCmAnodeConveyorPickUpBlower(enable := TRUE,   // "LBC_TwoWayActuatorCn"
                           parentReferenceDesignator := "Unit1.Em4.Config".em.referenceDesignator.combined,
                           enableManualCmds := #statEnableManualCmds,
                           interlockWorkPos := "Unit1.Em4.ControlNodes".cm.Interlock.anodeConveyorPickUpBlower.work,
                           interlockHomePos := "Unit1.Em4.ControlNodes".cm.Interlock.anodeConveyorPickUpBlower.home,
                           configuration := "Unit1.Em4.Config".cmAnodeConveyorPickUpBlower,
                           moduleInterface := "Unit1.Em4.HmiInterface".cmAnodeConveyorPickUpBlower,
                           controlNode := "Unit1.Em4.ControlNodes".cmAnodeConveyorPickUpBlower);
   "BA040AZSPM01.14" := #instCmAnodeConveyorPickUpBlower.goToWorkPos AND NOT #statUnitStatus.specialFunctions.dryRun;
END_REGION

REGION Network 283: ******************** Control Modules (Accessories) ********************
END_REGION

REGION Network 284: Reset CMS
   RUNG wire#powerrail
      Contact( #statUnitStatus.acknowledgeActive )
      wire#w1
      Contact( "Unit1.Em4.ControlNodes".cmAnodeVisionControllerInterface.monitoring.error )
      Coil( "Unit1.Em4.ControlNodes".cmAnodeVisionControllerInterface.commands.errorAck )
   END_RUNG
   RUNG wire#powerrail
      Contact( #statUnitStatus.state.resetting )
   END_RUNG wire#w1
   // the same network as SCL:
   "Unit1.Em4.ControlNodes".cmAnodeVisionControllerInterface.commands.errorAck := (#statUnitStatus.acknowledgeActive OR #statUnitStatus.state.resetting) AND "Unit1.Em4.ControlNodes".cmAnodeVisionControllerInterface.monitoring.error;
END_REGION

REGION Network 285: CmAnodeVisionControllerInterface Commands
   RUNG wire#powerrail
      I_Contact( "Unit1.Em4.ControlNodes".alignTable."step".action2[150] )
      I_Contact( "Unit1.Em4.ControlNodes".alignTable."step".action1[310] )
      Not()
      wire#w1
      Coil( "Unit1.Em4.ControlNodes".cmAnodeVisionControllerInterface.commands.stepStart )
   END_RUNG
   RUNG wire#powerrail
      I_Contact( "Unit1.Em4.ControlNodes".gaugeRnR."step".action1[610] )
      Not()
   END_RUNG wire#w1
   RUNG wire#powerrail
      I_Contact( "Unit1.MotionNodes".MotionToPLC.Status.OutputBits.AnodeAlignVision )
      Not()
   END_RUNG wire#w1
   // the same network as SCL:
   "Unit1.Em4.ControlNodes".cmAnodeVisionControllerInterface.commands.stepStart := NOT (NOT "Unit1.Em4.ControlNodes".alignTable."step".action2[150] AND NOT "Unit1.Em4.ControlNodes".alignTable."step".action1[310]) OR NOT (NOT "Unit1.Em4.ControlNodes".gaugeRnR."step".action1[610]) OR NOT (NOT "Unit1.MotionNodes".MotionToPLC.Status.OutputBits.AnodeAlignVision);
END_REGION

REGION Network 286: Call instCmAnodeVisionControllerInterface
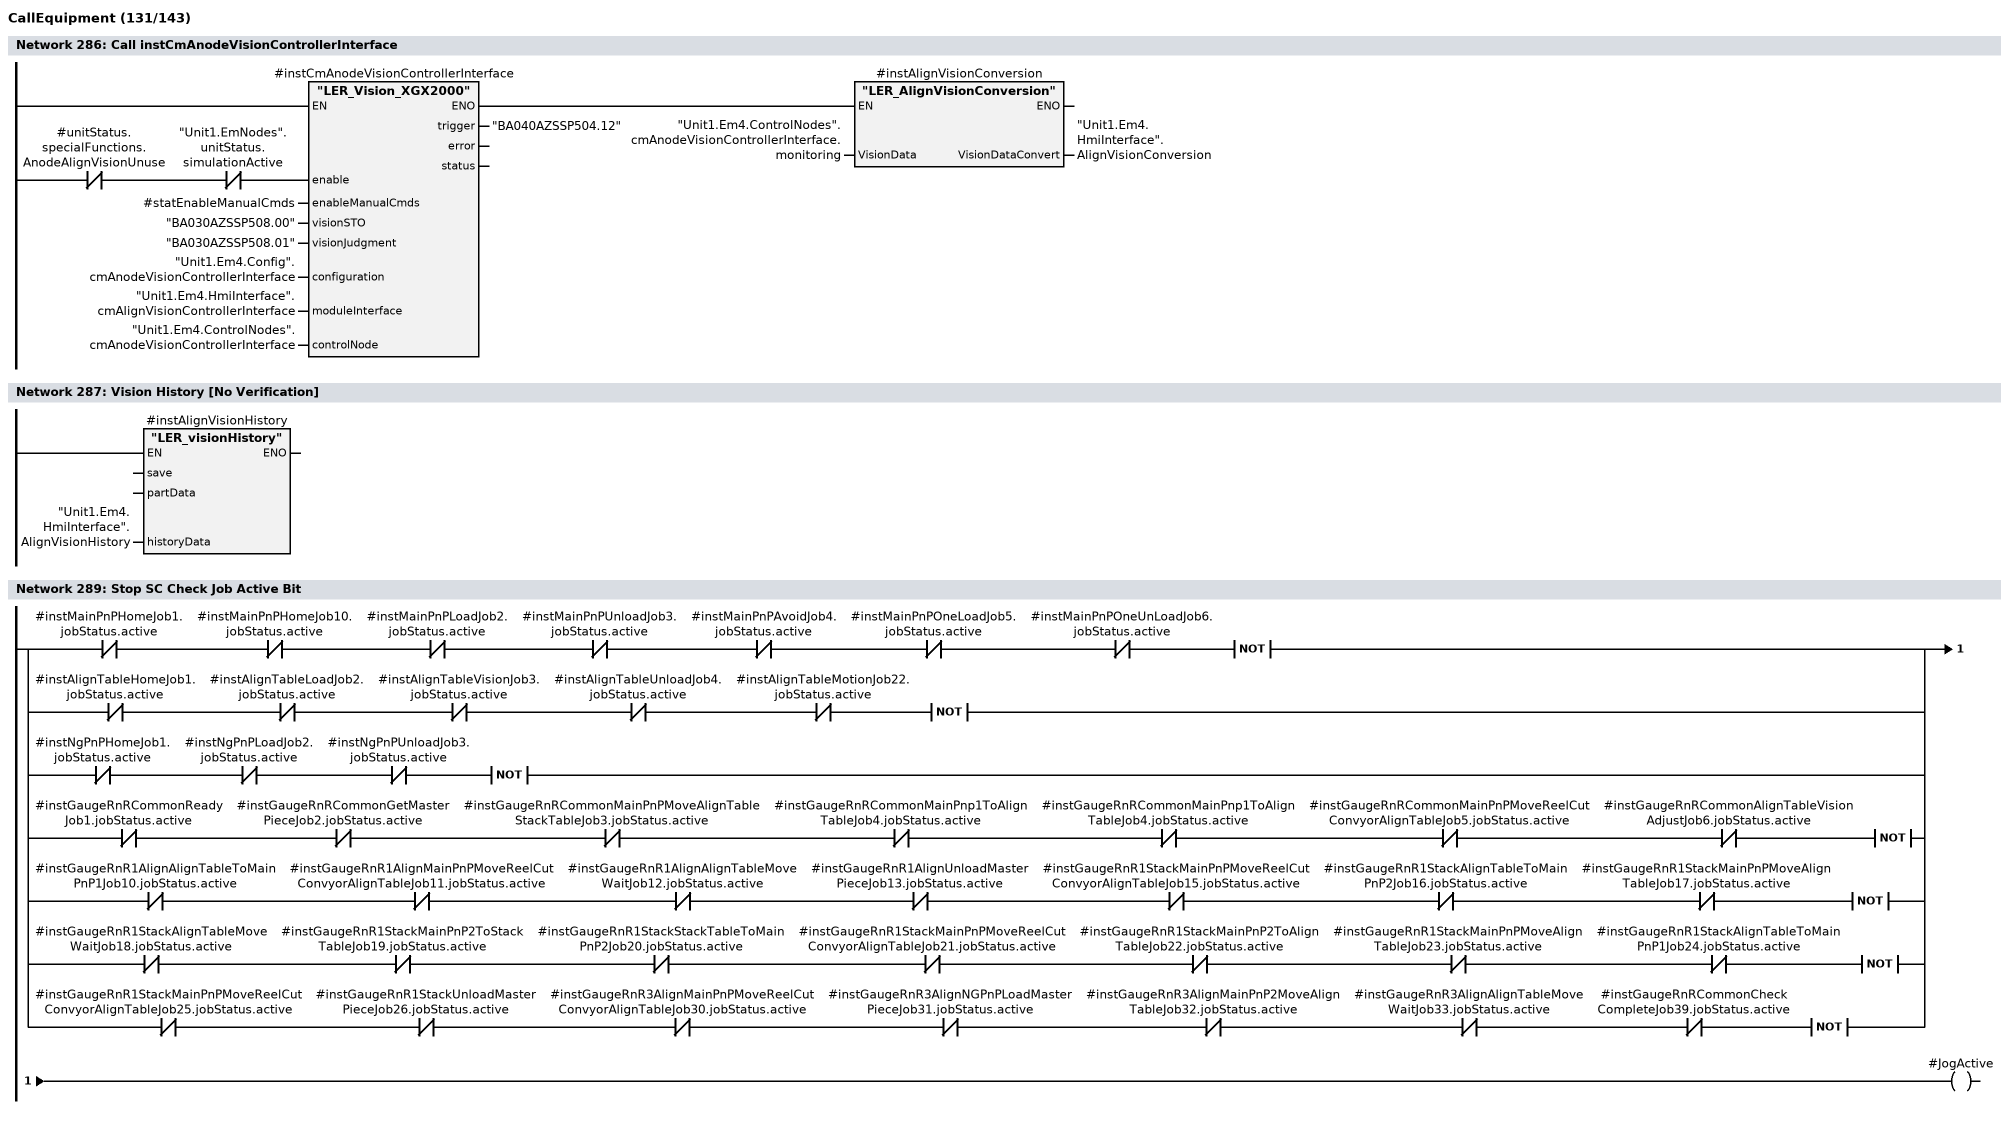
   RUNG wire#powerrail
      #instCmAnodeVisionControllerInterface(enable := wire#w1, enableManualCmds := #statEnableManualCmds, visionSTO := "BA030AZSSP508.00", visionJudgment := "BA030AZSSP508.01", configuration := "Unit1.Em4.Config".cmAnodeVisionControllerInterface, moduleInterface := "Unit1.Em4.HmiInterface".cmAlignVisionControllerInterface, controlNode := "Unit1.Em4.ControlNodes".cmAnodeVisionControllerInterface, trigger => "BA040AZSSP504.12", error =>, status =>)
      #instAlignVisionConversion(VisionData := "Unit1.Em4.ControlNodes".cmAnodeVisionControllerInterface.monitoring, VisionDataConvert => "Unit1.Em4.HmiInterface".AlignVisionConversion)
   END_RUNG
   RUNG wire#powerrail
      I_Contact( #unitStatus.specialFunctions.AnodeAlignVisionUnuse )
      I_Contact( "Unit1.EmNodes".unitStatus.simulationActive )
   END_RUNG wire#w1
   // the same network as SCL:
   #instCmAnodeVisionControllerInterface(enable := NOT #unitStatus.specialFunctions.AnodeAlignVisionUnuse AND NOT "Unit1.EmNodes".unitStatus.simulationActive,   // "LER_Vision_XGX2000"
                           enableManualCmds := #statEnableManualCmds,
                           visionSTO := "BA030AZSSP508.00",
                           visionJudgment := "BA030AZSSP508.01",
                           configuration := "Unit1.Em4.Config".cmAnodeVisionControllerInterface,
                           moduleInterface := "Unit1.Em4.HmiInterface".cmAlignVisionControllerInterface,
                           controlNode := "Unit1.Em4.ControlNodes".cmAnodeVisionControllerInterface,
                           trigger => "BA040AZSSP504.12",
                           ENO => #_w1);
   IF #_w1 THEN
       #instAlignVisionConversion(VisionData := "Unit1.Em4.ControlNodes".cmAnodeVisionControllerInterface.monitoring,   // "LER_AlignVisionConversion"
                               VisionDataConvert => "Unit1.Em4.HmiInterface".AlignVisionConversion);
   END_IF;
END_REGION

REGION Network 287: Vision History [No Verification]
   RUNG wire#powerrail
      #instAlignVisionHistory(save :=, partData :=, historyData := "Unit1.Em4.HmiInterface".AlignVisionHistory)
   END_RUNG
   // the same network as SCL:
   #instAlignVisionHistory(historyData := "Unit1.Em4.HmiInterface".AlignVisionHistory);   // "LER_visionHistory"
END_REGION

REGION Network 288: *************** Feedback to Unit ***************************
END_REGION

REGION Network 289: Stop SC Check Job Active Bit
   RUNG wire#powerrail
      I_Contact( #instMainPnPHomeJob1.jobStatus.active )
      I_Contact( #instMainPnPHomeJob10.jobStatus.active )
      I_Contact( #instMainPnPLoadJob2.jobStatus.active )
      I_Contact( #instMainPnPUnloadJob3.jobStatus.active )
      I_Contact( #instMainPnPAvoidJob4.jobStatus.active )
      I_Contact( #instMainPnPOneLoadJob5.jobStatus.active )
      I_Contact( #instMainPnPOneUnLoadJob6.jobStatus.active )
      Not()
      wire#w1
      Coil( #JogActive )
   END_RUNG
   RUNG wire#powerrail
      I_Contact( #instAlignTableHomeJob1.jobStatus.active )
      I_Contact( #instAlignTableLoadJob2.jobStatus.active )
      I_Contact( #instAlignTableVisionJob3.jobStatus.active )
      I_Contact( #instAlignTableUnloadJob4.jobStatus.active )
      I_Contact( #instAlignTableMotionJob22.jobStatus.active )
      Not()
   END_RUNG wire#w1
   RUNG wire#powerrail
      I_Contact( #instNgPnPHomeJob1.jobStatus.active )
      I_Contact( #instNgPnPLoadJob2.jobStatus.active )
      I_Contact( #instNgPnPUnloadJob3.jobStatus.active )
      Not()
   END_RUNG wire#w1
   RUNG wire#powerrail
      I_Contact( #instGaugeRnRCommonReadyJob1.jobStatus.active )
      I_Contact( #instGaugeRnRCommonGetMasterPieceJob2.jobStatus.active )
      I_Contact( #instGaugeRnRCommonMainPnPMoveAlignTableStackTableJob3.jobStatus.active )
      I_Contact( #instGaugeRnRCommonMainPnp1ToAlignTableJob4.jobStatus.active )
      I_Contact( #instGaugeRnRCommonMainPnp1ToAlignTableJob4.jobStatus.active )
      I_Contact( #instGaugeRnRCommonMainPnPMoveReelCutConvyorAlignTableJob5.jobStatus.active )
      I_Contact( #instGaugeRnRCommonAlignTableVisionAdjustJob6.jobStatus.active )
      Not()
   END_RUNG wire#w1
   RUNG wire#powerrail
      I_Contact( #instGaugeRnR1AlignAlignTableToMainPnP1Job10.jobStatus.active )
      I_Contact( #instGaugeRnR1AlignMainPnPMoveReelCutConvyorAlignTableJob11.jobStatus.active )
      I_Contact( #instGaugeRnR1AlignAlignTableMoveWaitJob12.jobStatus.active )
      I_Contact( #instGaugeRnR1AlignUnloadMasterPieceJob13.jobStatus.active )
      I_Contact( #instGaugeRnR1StackMainPnPMoveReelCutConvyorAlignTableJob15.jobStatus.active )
      I_Contact( #instGaugeRnR1StackAlignTableToMainPnP2Job16.jobStatus.active )
      I_Contact( #instGaugeRnR1StackMainPnPMoveAlignTableJob17.jobStatus.active )
      Not()
   END_RUNG wire#w1
   RUNG wire#powerrail
      I_Contact( #instGaugeRnR1StackAlignTableMoveWaitJob18.jobStatus.active )
      I_Contact( #instGaugeRnR1StackMainPnP2ToStackTableJob19.jobStatus.active )
      I_Contact( #instGaugeRnR1StackStackTableToMainPnP2Job20.jobStatus.active )
      I_Contact( #instGaugeRnR1StackMainPnPMoveReelCutConvyorAlignTableJob21.jobStatus.active )
      I_Contact( #instGaugeRnR1StackMainPnP2ToAlignTableJob22.jobStatus.active )
      I_Contact( #instGaugeRnR1StackMainPnPMoveAlignTableJob23.jobStatus.active )
      I_Contact( #instGaugeRnR1StackAlignTableToMainPnP1Job24.jobStatus.active )
      Not()
   END_RUNG wire#w1
   RUNG wire#powerrail
      I_Contact( #instGaugeRnR1StackMainPnPMoveReelCutConvyorAlignTableJob25.jobStatus.active )
      I_Contact( #instGaugeRnR1StackUnloadMasterPieceJob26.jobStatus.active )
      I_Contact( #instGaugeRnR3AlignMainPnPMoveReelCutConvyorAlignTableJob30.jobStatus.active )
      I_Contact( #instGaugeRnR3AlignNGPnPLoadMasterPieceJob31.jobStatus.active )
      I_Contact( #instGaugeRnR3AlignMainPnP2MoveAlignTableJob32.jobStatus.active )
      I_Contact( #instGaugeRnR3AlignAlignTableMoveWaitJob33.jobStatus.active )
      I_Contact( #instGaugeRnRCommonCheckCompleteJob39.jobStatus.active )
      Not()
   END_RUNG wire#w1
   // the same network as SCL:
   #JogActive := NOT (NOT #instMainPnPHomeJob1.jobStatus.active AND NOT #instMainPnPHomeJob10.jobStatus.active AND NOT #instMainPnPLoadJob2.jobStatus.active AND NOT #instMainPnPUnloadJob3.jobStatus.active AND NOT #instMainPnPAvoidJob4.jobStatus.active AND NOT #instMainPnPOneLoadJob5.jobStatus.active AND NOT #instMainPnPOneUnLoadJob6.jobStatus.active) OR NOT (NOT #instAlignTableHomeJob1.jobStatus.active AND NOT #instAlignTableLoadJob2.jobStatus.active AND NOT #instAlignTableVisionJob3.jobStatus.active AND NOT #instAlignTableUnloadJob4.jobStatus.active AND NOT #instAlignTableMotionJob22.jobStatus.active) OR NOT (NOT #instNgPnPHomeJob1.jobStatus.active AND NOT #instNgPnPLoadJob2.jobStatus.active AND NOT #instNgPnPUnloadJob3.jobStatus.active) OR NOT (NOT #instGaugeRnRCommonReadyJob1.jobStatus.active AND NOT #instGaugeRnRCommonGetMasterPieceJob2.jobStatus.active AND NOT #instGaugeRnRCommonMainPnPMoveAlignTableStackTableJob3.jobStatus.active AND NOT #instGaugeRnRCommonMainPnp1ToAlignTableJob4.jobStatus.active AND NOT #instGaugeRnRCommonMainPnp1ToAlignTableJob4.jobStatus.active AND NOT #instGaugeRnRCommonMainPnPMoveReelCutConvyorAlignTableJob5.jobStatus.active AND NOT #instGaugeRnRCommonAlignTableVisionAdjustJob6.jobStatus.active) OR NOT (NOT #instGaugeRnR1AlignAlignTableToMainPnP1Job10.jobStatus.active AND NOT #instGaugeRnR1AlignMainPnPMoveReelCutConvyorAlignTableJob11.jobStatus.active AND NOT #instGaugeRnR1AlignAlignTableMoveWaitJob12.jobStatus.active AND NOT #instGaugeRnR1AlignUnloadMasterPieceJob13.jobStatus.active AND NOT #instGaugeRnR1StackMainPnPMoveReelCutConvyorAlignTableJob15.jobStatus.active AND NOT #instGaugeRnR1StackAlignTableToMainPnP2Job16.jobStatus.active AND NOT #instGaugeRnR1StackMainPnPMoveAlignTableJob17.jobStatus.active) OR NOT (NOT #instGaugeRnR1StackAlignTableMoveWaitJob18.jobStatus.active AND NOT #instGaugeRnR1StackMainPnP2ToStackTableJob19.jobStatus.active AND NOT #instGaugeRnR1StackStackTableToMainPnP2Job20.jobStatus.active AND NOT #instGaugeRnR1StackMainPnPMoveReelCutConvyorAlignTableJob21.jobStatus.active AND NOT #instGaugeRnR1StackMainPnP2ToAlignTableJob22.jobStatus.active AND NOT #instGaugeRnR1StackMainPnPMoveAlignTableJob23.jobStatus.active AND NOT #instGaugeRnR1StackAlignTableToMainPnP1Job24.jobStatus.active) OR NOT (NOT #instGaugeRnR1StackMainPnPMoveReelCutConvyorAlignTableJob25.jobStatus.active AND NOT #instGaugeRnR1StackUnloadMasterPieceJob26.jobStatus.active AND NOT #instGaugeRnR3AlignMainPnPMoveReelCutConvyorAlignTableJob30.jobStatus.active AND NOT #instGaugeRnR3AlignNGPnPLoadMasterPieceJob31.jobStatus.active AND NOT #instGaugeRnR3AlignMainPnP2MoveAlignTableJob32.jobStatus.active AND NOT #instGaugeRnR3AlignAlignTableMoveWaitJob33.jobStatus.active AND NOT #instGaugeRnRCommonCheckCompleteJob39.jobStatus.active);
END_REGION

REGION Network 290: Determine StateComplete (SC) in Mode Production
   // Conditions for the Equipment Modules "stateComplete" feedback to the unit. This feedback is given when the task in for the respective state is complete.
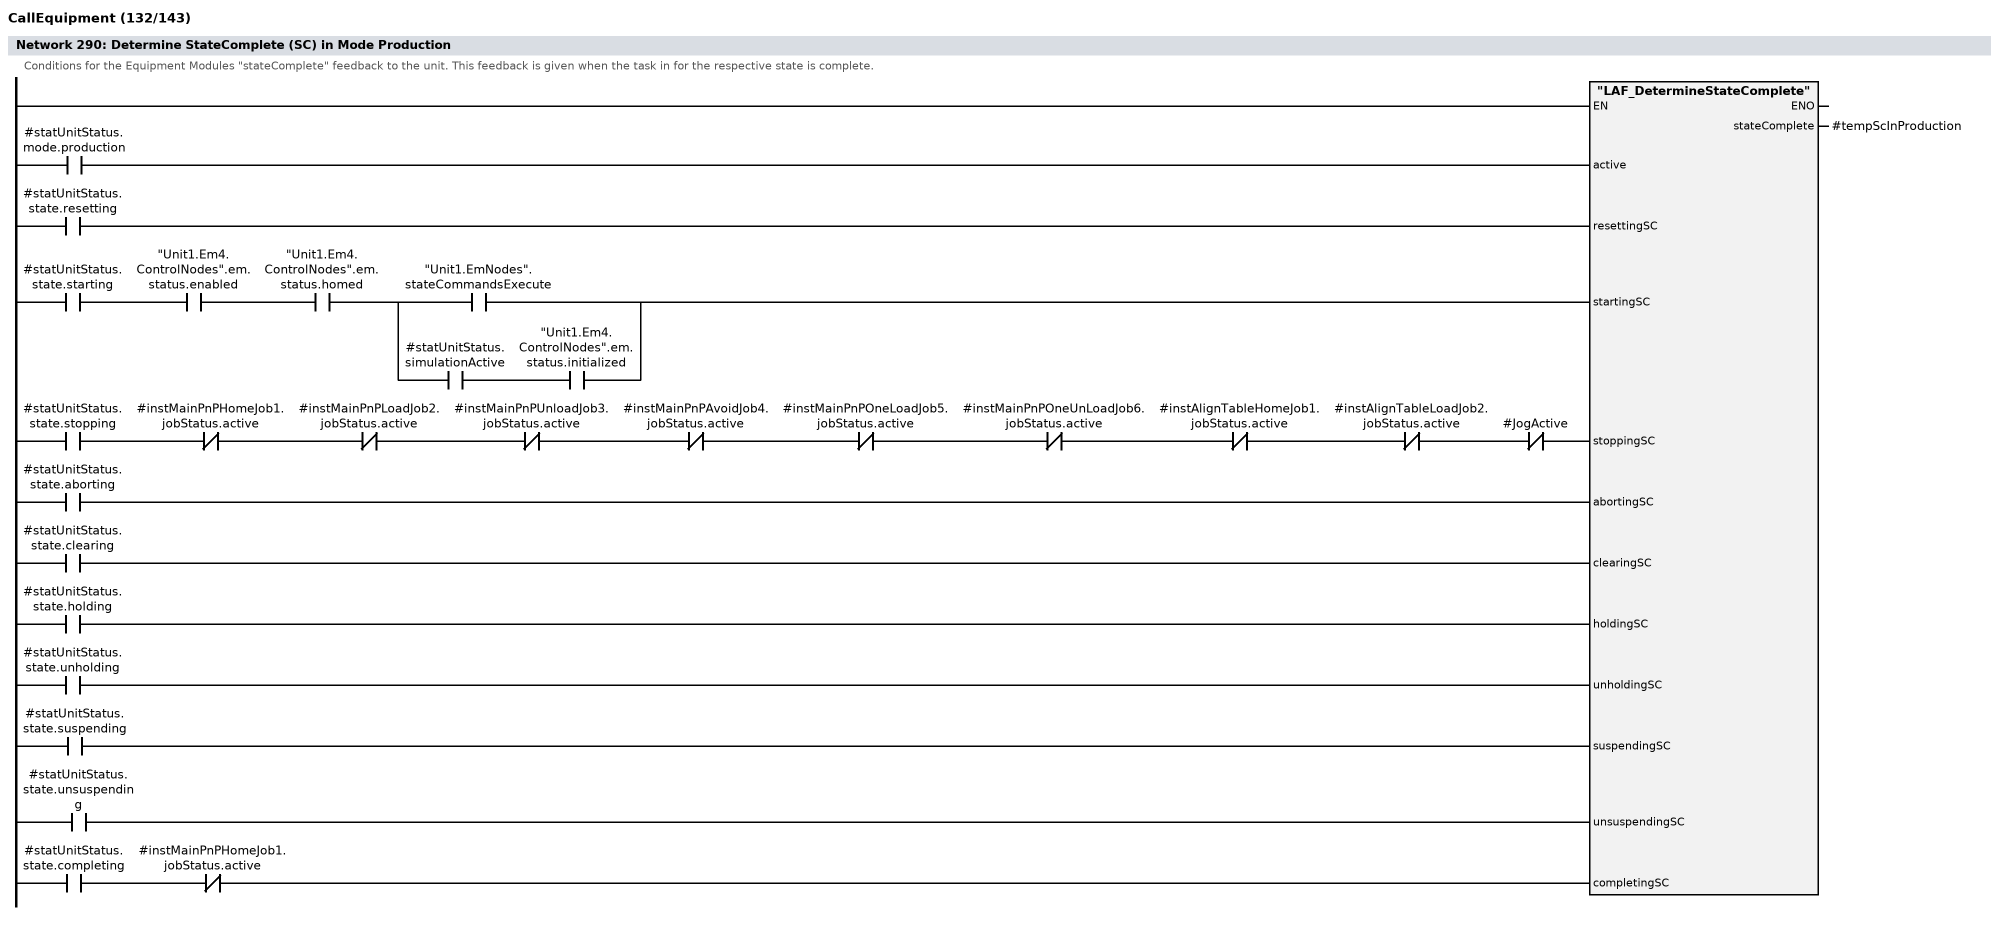
   RUNG wire#powerrail
      "LAF_DetermineStateComplete"(active := wire#w1, resettingSC := wire#w2, startingSC := wire#w4, stoppingSC := wire#w5, abortingSC := wire#w6, clearingSC := wire#w7, holdingSC := wire#w8, unholdingSC := wire#w9, suspendingSC := wire#w10, unsuspendingSC := wire#w11, completingSC := wire#w12, stateComplete => #tempScInProduction)
   END_RUNG
   RUNG wire#powerrail
      Contact( #statUnitStatus.mode.production )
   END_RUNG wire#w1
   RUNG wire#powerrail
      Contact( #statUnitStatus.state.resetting )
   END_RUNG wire#w2
   RUNG wire#powerrail
      Contact( #statUnitStatus.state.starting )
      Contact( "Unit1.Em4.ControlNodes".em.status.enabled )
      Contact( "Unit1.Em4.ControlNodes".em.status.homed )
      wire#w3
      Contact( "Unit1.EmNodes".stateCommandsExecute )
   END_RUNG wire#w4
   RUNG wire#w3
      Contact( #statUnitStatus.simulationActive )
      Contact( "Unit1.Em4.ControlNodes".em.status.initialized )
   END_RUNG wire#w4
   RUNG wire#powerrail
      Contact( #statUnitStatus.state.stopping )
      I_Contact( #instMainPnPHomeJob1.jobStatus.active )
      I_Contact( #instMainPnPLoadJob2.jobStatus.active )
      I_Contact( #instMainPnPUnloadJob3.jobStatus.active )
      I_Contact( #instMainPnPAvoidJob4.jobStatus.active )
      I_Contact( #instMainPnPOneLoadJob5.jobStatus.active )
      I_Contact( #instMainPnPOneUnLoadJob6.jobStatus.active )
      I_Contact( #instAlignTableHomeJob1.jobStatus.active )
      I_Contact( #instAlignTableLoadJob2.jobStatus.active )
      I_Contact( #JogActive )
   END_RUNG wire#w5
   RUNG wire#powerrail
      Contact( #statUnitStatus.state.aborting )
   END_RUNG wire#w6
   RUNG wire#powerrail
      Contact( #statUnitStatus.state.clearing )
   END_RUNG wire#w7
   RUNG wire#powerrail
      Contact( #statUnitStatus.state.holding )
   END_RUNG wire#w8
   RUNG wire#powerrail
      Contact( #statUnitStatus.state.unholding )
   END_RUNG wire#w9
   RUNG wire#powerrail
      Contact( #statUnitStatus.state.suspending )
   END_RUNG wire#w10
   RUNG wire#powerrail
      Contact( #statUnitStatus.state.unsuspending )
   END_RUNG wire#w11
   RUNG wire#powerrail
      Contact( #statUnitStatus.state.completing )
      I_Contact( #instMainPnPHomeJob1.jobStatus.active )
   END_RUNG wire#w12
   // the same network as SCL:
   "LAF_DetermineStateComplete"(active := #statUnitStatus.mode.production,
                           resettingSC := #statUnitStatus.state.resetting,
                           startingSC := #statUnitStatus.state.starting AND "Unit1.Em4.ControlNodes".em.status.enabled AND "Unit1.Em4.ControlNodes".em.status.homed AND ("Unit1.EmNodes".stateCommandsExecute OR (#statUnitStatus.simulationActive AND "Unit1.Em4.ControlNodes".em.status.initialized)),
                           stoppingSC := #statUnitStatus.state.stopping AND NOT #instMainPnPHomeJob1.jobStatus.active AND NOT #instMainPnPLoadJob2.jobStatus.active AND NOT #instMainPnPUnloadJob3.jobStatus.active AND NOT #instMainPnPAvoidJob4.jobStatus.active AND NOT #instMainPnPOneLoadJob5.jobStatus.active AND NOT #instMainPnPOneUnLoadJob6.jobStatus.active AND NOT #instAlignTableHomeJob1.jobStatus.active AND NOT #instAlignTableLoadJob2.jobStatus.active AND NOT #JogActive,
                           abortingSC := #statUnitStatus.state.aborting,
                           clearingSC := #statUnitStatus.state.clearing,
                           holdingSC := #statUnitStatus.state.holding,
                           unholdingSC := #statUnitStatus.state.unholding,
                           suspendingSC := #statUnitStatus.state.suspending,
                           unsuspendingSC := #statUnitStatus.state.unsuspending,
                           completingSC := #statUnitStatus.state.completing AND NOT #instMainPnPHomeJob1.jobStatus.active,
                           stateComplete => #tempScInProduction);
END_REGION

REGION Network 291: Determine StateComplete (SC) in Mode Maintenance/Manual
   // Conditions for the Equipment Modules "stateComplete" feedback to the unit. This feedback is given when the task in for the respective state is complete.
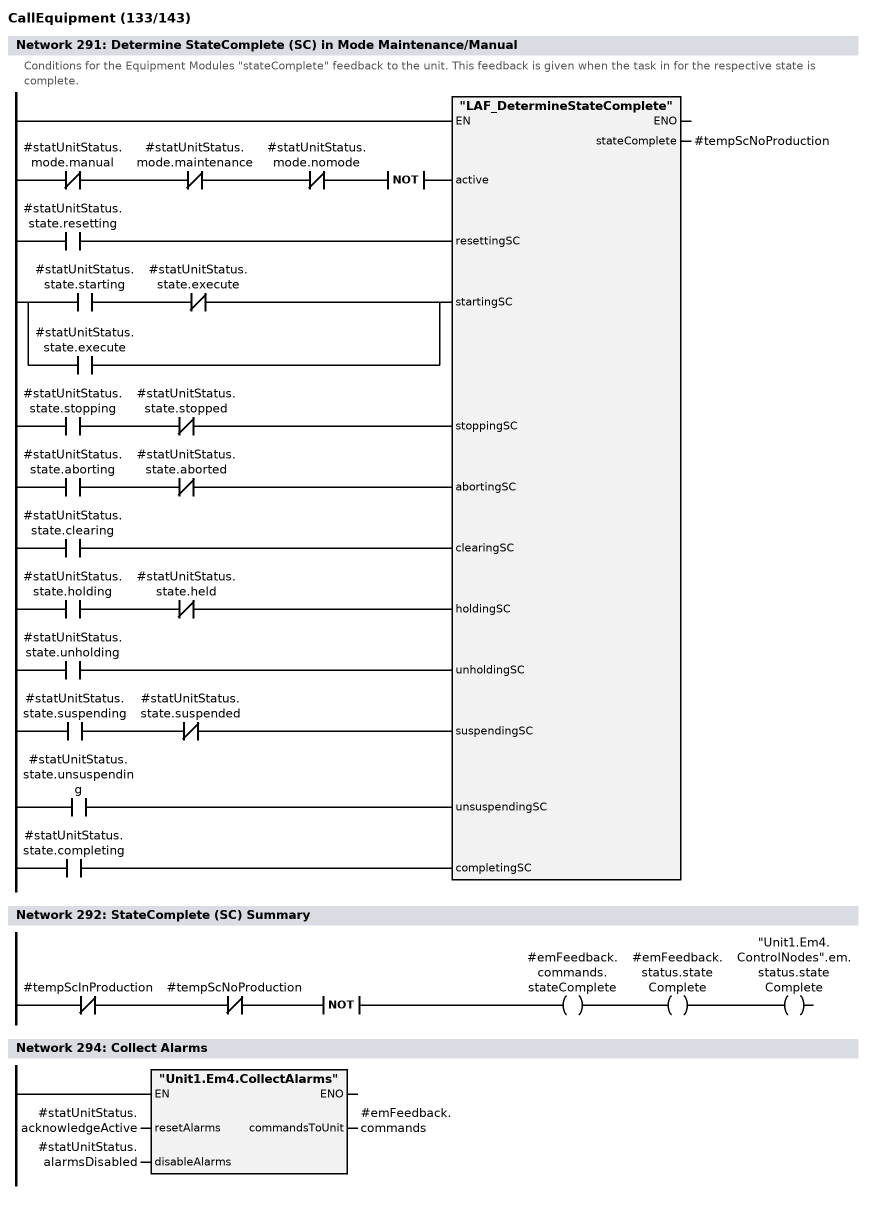
   RUNG wire#powerrail
      "LAF_DetermineStateComplete"(active := wire#w1, resettingSC := wire#w2, startingSC := wire#w3, stoppingSC := wire#w4, abortingSC := wire#w5, clearingSC := wire#w6, holdingSC := wire#w7, unholdingSC := wire#w8, suspendingSC := wire#w9, unsuspendingSC := wire#w10, completingSC := wire#w11, stateComplete => #tempScNoProduction)
   END_RUNG
   RUNG wire#powerrail
      I_Contact( #statUnitStatus.mode.manual )
      I_Contact( #statUnitStatus.mode.maintenance )
      I_Contact( #statUnitStatus.mode.nomode )
      Not()
   END_RUNG wire#w1
   RUNG wire#powerrail
      Contact( #statUnitStatus.state.resetting )
   END_RUNG wire#w2
   RUNG wire#powerrail
      Contact( #statUnitStatus.state.starting )
      I_Contact( #statUnitStatus.state.execute )
   END_RUNG wire#w3
   RUNG wire#powerrail
      Contact( #statUnitStatus.state.execute )
   END_RUNG wire#w3
   RUNG wire#powerrail
      Contact( #statUnitStatus.state.stopping )
      I_Contact( #statUnitStatus.state.stopped )
   END_RUNG wire#w4
   RUNG wire#powerrail
      Contact( #statUnitStatus.state.aborting )
      I_Contact( #statUnitStatus.state.aborted )
   END_RUNG wire#w5
   RUNG wire#powerrail
      Contact( #statUnitStatus.state.clearing )
   END_RUNG wire#w6
   RUNG wire#powerrail
      Contact( #statUnitStatus.state.holding )
      I_Contact( #statUnitStatus.state.held )
   END_RUNG wire#w7
   RUNG wire#powerrail
      Contact( #statUnitStatus.state.unholding )
   END_RUNG wire#w8
   RUNG wire#powerrail
      Contact( #statUnitStatus.state.suspending )
      I_Contact( #statUnitStatus.state.suspended )
   END_RUNG wire#w9
   RUNG wire#powerrail
      Contact( #statUnitStatus.state.unsuspending )
   END_RUNG wire#w10
   RUNG wire#powerrail
      Contact( #statUnitStatus.state.completing )
   END_RUNG wire#w11
   // the same network as SCL:
   "LAF_DetermineStateComplete"(active := NOT (NOT #statUnitStatus.mode.manual AND NOT #statUnitStatus.mode.maintenance AND NOT #statUnitStatus.mode.nomode),
                           resettingSC := #statUnitStatus.state.resetting,
                           startingSC := (#statUnitStatus.state.starting AND NOT #statUnitStatus.state.execute) OR #statUnitStatus.state.execute,
                           stoppingSC := #statUnitStatus.state.stopping AND NOT #statUnitStatus.state.stopped,
                           abortingSC := #statUnitStatus.state.aborting AND NOT #statUnitStatus.state.aborted,
                           clearingSC := #statUnitStatus.state.clearing,
                           holdingSC := #statUnitStatus.state.holding AND NOT #statUnitStatus.state.held,
                           unholdingSC := #statUnitStatus.state.unholding,
                           suspendingSC := #statUnitStatus.state.suspending AND NOT #statUnitStatus.state.suspended,
                           unsuspendingSC := #statUnitStatus.state.unsuspending,
                           completingSC := #statUnitStatus.state.completing,
                           stateComplete => #tempScNoProduction);
END_REGION

REGION Network 292: StateComplete (SC) Summary
   RUNG wire#powerrail
      I_Contact( #tempScInProduction )
      I_Contact( #tempScNoProduction )
      Not()
      Coil( #emFeedback.commands.stateComplete )
      Coil( #emFeedback.status.stateComplete )
      Coil( "Unit1.Em4.ControlNodes".em.status.stateComplete )
   END_RUNG
   // the same network as SCL:
   #emFeedback.commands.stateComplete := NOT (NOT #tempScInProduction AND NOT #tempScNoProduction);
   #emFeedback.status.stateComplete := #emFeedback.commands.stateComplete;
   "Unit1.Em4.ControlNodes".em.status.stateComplete := #emFeedback.commands.stateComplete;
END_REGION

REGION Network 293: *************** Alarms **********************************
END_REGION

REGION Network 294: Collect Alarms
   RUNG wire#powerrail
      "Unit1.Em4.CollectAlarms"(resetAlarms := #statUnitStatus.acknowledgeActive, disableAlarms := #statUnitStatus.alarmsDisabled, commandsToUnit => #emFeedback.commands)
   END_RUNG
   // the same network as SCL:
   "Unit1.Em4.CollectAlarms"(resetAlarms := #statUnitStatus.acknowledgeActive,
                           disableAlarms := #statUnitStatus.alarmsDisabled,
                           commandsToUnit => #emFeedback.commands);
END_REGION

REGION Network 295: Manage Alarms
   // Derive commands from the ProDiag supervision. The ProDiag supervisions contain categories which define the reaction of these supervisions (e.g. abort, stop, hold). These are handed over as commands to the unit level.
   // Alternatively, if no ProDiag should be used, you can use the LAF_ManageBitAlarms to realize bit alarm handling. This block can be found in LAF in folder 70_AlarmHandling.
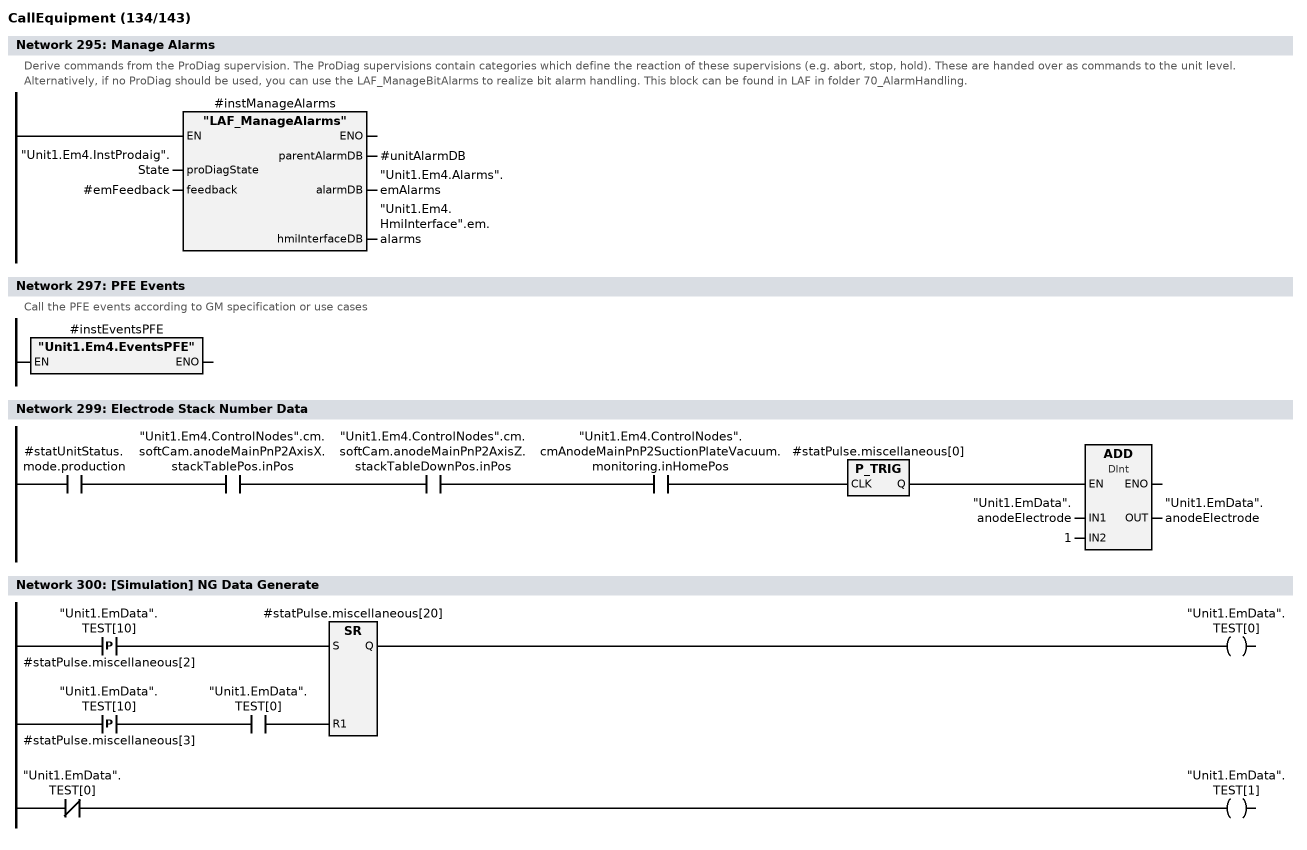
   RUNG wire#powerrail
      #instManageAlarms(proDiagState := "Unit1.Em4.InstProdaig".State, feedback := #emFeedback, parentAlarmDB => #unitAlarmDB, alarmDB => "Unit1.Em4.Alarms".emAlarms, hmiInterfaceDB => "Unit1.Em4.HmiInterface".em.alarms)
   END_RUNG
   // the same network as SCL:
   #instManageAlarms(proDiagState := "Unit1.Em4.InstProdaig".State,   // "LAF_ManageAlarms"
                     feedback := #emFeedback,
                     parentAlarmDB => #unitAlarmDB,
                     alarmDB => "Unit1.Em4.Alarms".emAlarms,
                     hmiInterfaceDB => "Unit1.Em4.HmiInterface".em.alarms);
END_REGION

REGION Network 296: *************** PFE Events**********************************
END_REGION

REGION Network 297: PFE Events
   // Call the PFE events according to GM specification or use cases
   RUNG wire#powerrail
      #instEventsPFE()
   END_RUNG
   // the same network as SCL:
   #instEventsPFE();   // "Unit1.Em4.EventsPFE"
END_REGION

REGION Network 298: ******************** Part Data ********************
END_REGION

REGION Network 299: Electrode Stack Number Data
   RUNG wire#powerrail
      Contact( #statUnitStatus.mode.production )
      Contact( "Unit1.Em4.ControlNodes".cm.softCam.anodeMainPnP2AxisX.stackTablePos.inPos )
      Contact( "Unit1.Em4.ControlNodes".cm.softCam.anodeMainPnP2AxisZ.stackTableDownPos.inPos )
      Contact( "Unit1.Em4.ControlNodes".cmAnodeMainPnP2SuctionPlateVacuum.monitoring.inHomePos )
      P_Trig( #statPulse.miscellaneous[0] )
      { S7_Templates := "SrcType := DInt" } Add(in1 := "Unit1.EmData".anodeElectrode, in2 := 1, out => "Unit1.EmData".anodeElectrode)
   END_RUNG
   // the same network as SCL:
   #_w1 := #statUnitStatus.mode.production AND "Unit1.Em4.ControlNodes".cm.softCam.anodeMainPnP2AxisX.stackTablePos.inPos AND "Unit1.Em4.ControlNodes".cm.softCam.anodeMainPnP2AxisZ.stackTableDownPos.inPos AND "Unit1.Em4.ControlNodes".cmAnodeMainPnP2SuctionPlateVacuum.monitoring.inHomePos;
   #_w2 := #_w1 AND NOT #statPulse.miscellaneous[0];   // rising edge
   #statPulse.miscellaneous[0] := #_w1;
   IF #_w2 THEN "Unit1.EmData".anodeElectrode := "Unit1.EmData".anodeElectrode + 1; END_IF;
END_REGION

REGION Network 300: [Simulation] NG Data Generate
   RUNG wire#powerrail
      P_Contact(operand := "Unit1.EmData".TEST[10], bit := #statPulse.miscellaneous[2])
      S_SR(operand := #statPulse.miscellaneous[20], r1 := wire#w1)
      Coil( "Unit1.EmData".TEST[0] )
   END_RUNG
   RUNG wire#powerrail
      P_Contact(operand := "Unit1.EmData".TEST[10], bit := #statPulse.miscellaneous[3])
      Contact( "Unit1.EmData".TEST[0] )
   END_RUNG wire#w1
   RUNG wire#powerrail
      I_Contact( "Unit1.EmData".TEST[0] )
      Coil( "Unit1.EmData".TEST[1] )
   END_RUNG
   // the same network as SCL:
   #_w1 := "Unit1.EmData".TEST[10] AND NOT #statPulse.miscellaneous[2];   // rising edge of "Unit1.EmData".TEST[10]
   #statPulse.miscellaneous[2] := "Unit1.EmData".TEST[10];
   #_w2 := "Unit1.EmData".TEST[10] AND NOT #statPulse.miscellaneous[3];   // rising edge of "Unit1.EmData".TEST[10]
   #statPulse.miscellaneous[3] := "Unit1.EmData".TEST[10];
   IF #_w1 THEN
       #statPulse.miscellaneous[20] := TRUE;   // SR flip-flop
   END_IF;
   IF #_w2 AND "Unit1.EmData".TEST[0] THEN #statPulse.miscellaneous[20] := FALSE; END_IF;
   "Unit1.EmData".TEST[0] := #statPulse.miscellaneous[20];
   "Unit1.EmData".TEST[1] := NOT "Unit1.EmData".TEST[0];
END_REGION

REGION Network 301: Align Vision Data
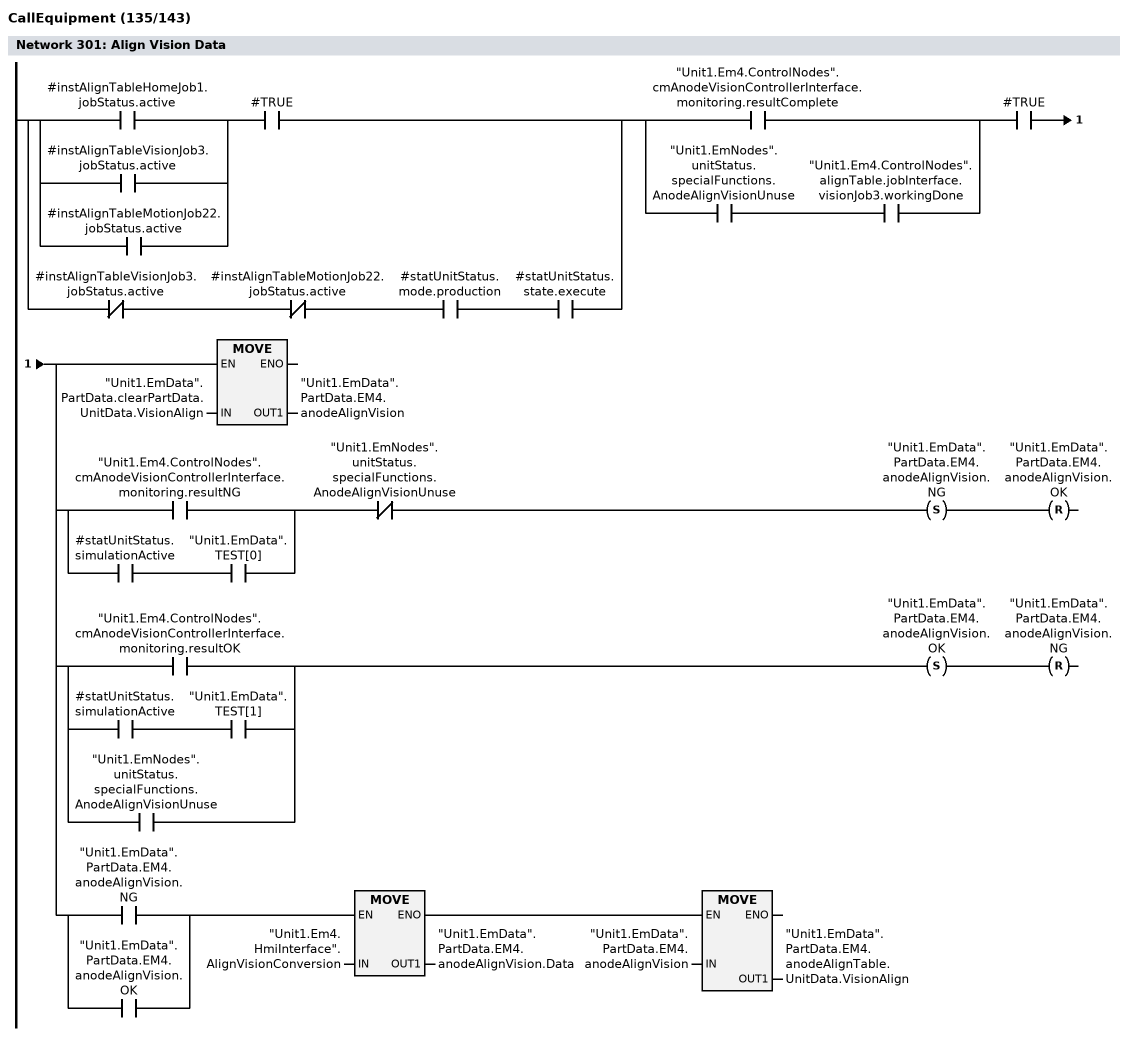
   RUNG wire#powerrail
      Contact( #instAlignTableHomeJob1.jobStatus.active )
      wire#w1
      Contact( #TRUE )
      wire#w2
      Contact( "Unit1.Em4.ControlNodes".cmAnodeVisionControllerInterface.monitoring.resultComplete )
      wire#w3
      Contact( #TRUE )
      wire#w4
      Move(in := "Unit1.EmData".PartData.clearPartData.UnitData.VisionAlign, out1 => "Unit1.EmData".PartData.EM4.anodeAlignVision)
   END_RUNG
   RUNG wire#powerrail
      Contact( #instAlignTableVisionJob3.jobStatus.active )
   END_RUNG wire#w1
   RUNG wire#powerrail
      Contact( #instAlignTableMotionJob22.jobStatus.active )
   END_RUNG wire#w1
   RUNG wire#powerrail
      I_Contact( #instAlignTableVisionJob3.jobStatus.active )
      I_Contact( #instAlignTableMotionJob22.jobStatus.active )
      Contact( #statUnitStatus.mode.production )
      Contact( #statUnitStatus.state.execute )
   END_RUNG wire#w2
   RUNG wire#w2
      Contact( "Unit1.EmNodes".unitStatus.specialFunctions.AnodeAlignVisionUnuse )
      Contact( "Unit1.Em4.ControlNodes".alignTable.jobInterface.visionJob3.workingDone )
   END_RUNG wire#w3
   RUNG wire#w4
      Contact( "Unit1.Em4.ControlNodes".cmAnodeVisionControllerInterface.monitoring.resultNG )
      wire#w5
      I_Contact( "Unit1.EmNodes".unitStatus.specialFunctions.AnodeAlignVisionUnuse )
      S_Coil( "Unit1.EmData".PartData.EM4.anodeAlignVision.NG )
      R_Coil( "Unit1.EmData".PartData.EM4.anodeAlignVision.OK )
   END_RUNG
   RUNG wire#w4
      Contact( #statUnitStatus.simulationActive )
      Contact( "Unit1.EmData".TEST[0] )
   END_RUNG wire#w5
   RUNG wire#w4
      Contact( "Unit1.Em4.ControlNodes".cmAnodeVisionControllerInterface.monitoring.resultOK )
      wire#w6
      S_Coil( "Unit1.EmData".PartData.EM4.anodeAlignVision.OK )
      R_Coil( "Unit1.EmData".PartData.EM4.anodeAlignVision.NG )
   END_RUNG
   RUNG wire#w4
      Contact( #statUnitStatus.simulationActive )
      Contact( "Unit1.EmData".TEST[1] )
   END_RUNG wire#w6
   RUNG wire#w4
      Contact( "Unit1.EmNodes".unitStatus.specialFunctions.AnodeAlignVisionUnuse )
   END_RUNG wire#w6
   RUNG wire#w4
      Contact( "Unit1.EmData".PartData.EM4.anodeAlignVision.NG )
      wire#w7
      Move(in := "Unit1.Em4.HmiInterface".AlignVisionConversion, out1 => "Unit1.EmData".PartData.EM4.anodeAlignVision.Data)
      Move(in := "Unit1.EmData".PartData.EM4.anodeAlignVision, out1 => "Unit1.EmData".PartData.EM4.anodeAlignTable.UnitData.VisionAlign)
   END_RUNG
   RUNG wire#w4
      Contact( "Unit1.EmData".PartData.EM4.anodeAlignVision.OK )
   END_RUNG wire#w7
   // the same network as SCL:
   #_w1 := (((#instAlignTableHomeJob1.jobStatus.active OR #instAlignTableVisionJob3.jobStatus.active OR #instAlignTableMotionJob22.jobStatus.active) AND #TRUE) OR (NOT #instAlignTableVisionJob3.jobStatus.active AND NOT #instAlignTableMotionJob22.jobStatus.active AND #statUnitStatus.mode.production AND #statUnitStatus.state.execute)) AND ("Unit1.Em4.ControlNodes".cmAnodeVisionControllerInterface.monitoring.resultComplete OR ("Unit1.EmNodes".unitStatus.specialFunctions.AnodeAlignVisionUnuse AND "Unit1.Em4.ControlNodes".alignTable.jobInterface.visionJob3.workingDone)) AND #TRUE;
   IF #_w1 THEN
       "Unit1.EmData".PartData.EM4.anodeAlignVision := "Unit1.EmData".PartData.clearPartData.UnitData.VisionAlign;
   END_IF;
   IF #_w1 AND ("Unit1.Em4.ControlNodes".cmAnodeVisionControllerInterface.monitoring.resultNG OR (#statUnitStatus.simulationActive AND "Unit1.EmData".TEST[0])) AND NOT "Unit1.EmNodes".unitStatus.specialFunctions.AnodeAlignVisionUnuse THEN
       "Unit1.EmData".PartData.EM4.anodeAlignVision.NG := TRUE;
       "Unit1.EmData".PartData.EM4.anodeAlignVision.OK := FALSE;
   END_IF;
   IF #_w1 AND ("Unit1.Em4.ControlNodes".cmAnodeVisionControllerInterface.monitoring.resultOK OR (#statUnitStatus.simulationActive AND "Unit1.EmData".TEST[1]) OR "Unit1.EmNodes".unitStatus.specialFunctions.AnodeAlignVisionUnuse) THEN
       "Unit1.EmData".PartData.EM4.anodeAlignVision.OK := TRUE;
       "Unit1.EmData".PartData.EM4.anodeAlignVision.NG := FALSE;
   END_IF;
   IF #_w1 AND ("Unit1.EmData".PartData.EM4.anodeAlignVision.NG OR "Unit1.EmData".PartData.EM4.anodeAlignVision.OK) THEN
       "Unit1.EmData".PartData.EM4.anodeAlignVision.Data := "Unit1.Em4.HmiInterface".AlignVisionConversion;
       "Unit1.EmData".PartData.EM4.anodeAlignTable.UnitData.VisionAlign := "Unit1.EmData".PartData.EM4.anodeAlignVision;
   END_IF;
END_REGION

REGION Network 302: ******************** Unit Output ********************
END_REGION

REGION Network 303 (SCL): Sync Motion
   // Em → Unit1 Mapping
END_REGION

REGION Network 304: Em Nodes Brake Test
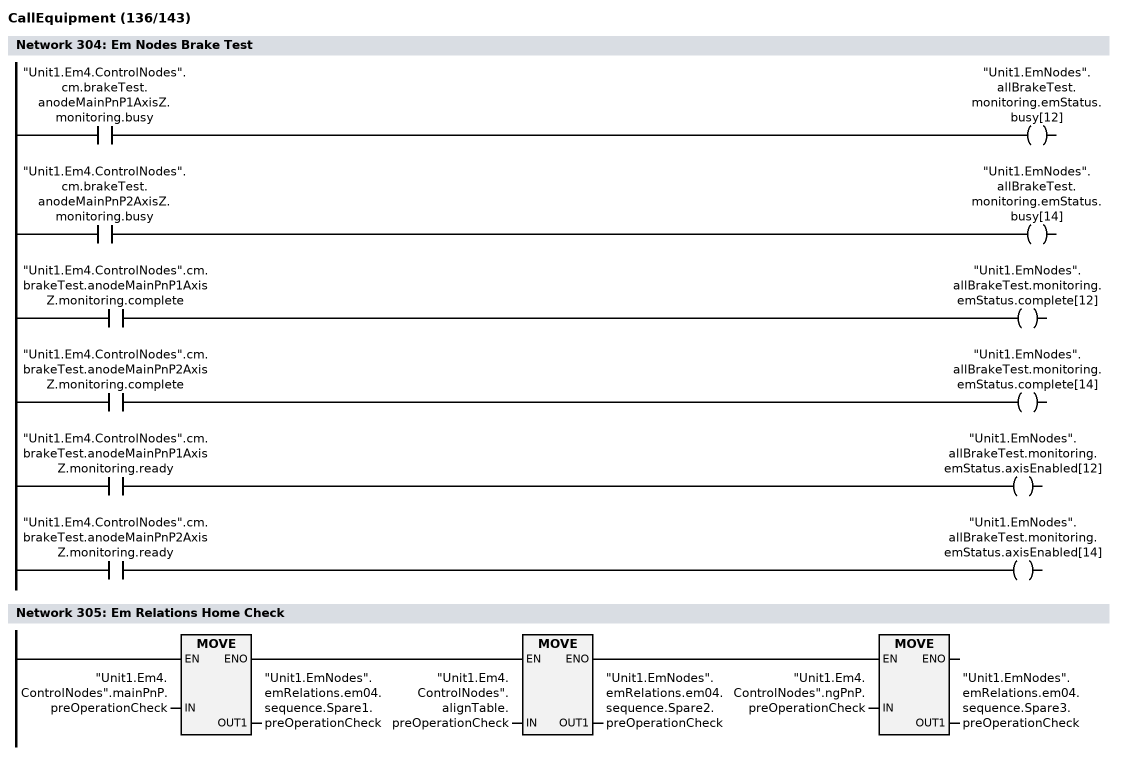
   RUNG wire#powerrail
      Contact( "Unit1.Em4.ControlNodes".cm.brakeTest.anodeMainPnP1AxisZ.monitoring.busy )
      Coil( "Unit1.EmNodes".allBrakeTest.monitoring.emStatus.busy[12] )
   END_RUNG
   RUNG wire#powerrail
      Contact( "Unit1.Em4.ControlNodes".cm.brakeTest.anodeMainPnP2AxisZ.monitoring.busy )
      Coil( "Unit1.EmNodes".allBrakeTest.monitoring.emStatus.busy[14] )
   END_RUNG
   RUNG wire#powerrail
      Contact( "Unit1.Em4.ControlNodes".cm.brakeTest.anodeMainPnP1AxisZ.monitoring.complete )
      Coil( "Unit1.EmNodes".allBrakeTest.monitoring.emStatus.complete[12] )
   END_RUNG
   RUNG wire#powerrail
      Contact( "Unit1.Em4.ControlNodes".cm.brakeTest.anodeMainPnP2AxisZ.monitoring.complete )
      Coil( "Unit1.EmNodes".allBrakeTest.monitoring.emStatus.complete[14] )
   END_RUNG
   RUNG wire#powerrail
      Contact( "Unit1.Em4.ControlNodes".cm.brakeTest.anodeMainPnP1AxisZ.monitoring.ready )
      Coil( "Unit1.EmNodes".allBrakeTest.monitoring.emStatus.axisEnabled[12] )
   END_RUNG
   RUNG wire#powerrail
      Contact( "Unit1.Em4.ControlNodes".cm.brakeTest.anodeMainPnP2AxisZ.monitoring.ready )
      Coil( "Unit1.EmNodes".allBrakeTest.monitoring.emStatus.axisEnabled[14] )
   END_RUNG
   // the same network as SCL:
   "Unit1.EmNodes".allBrakeTest.monitoring.emStatus.busy[12] := "Unit1.Em4.ControlNodes".cm.brakeTest.anodeMainPnP1AxisZ.monitoring.busy;
   "Unit1.EmNodes".allBrakeTest.monitoring.emStatus.busy[14] := "Unit1.Em4.ControlNodes".cm.brakeTest.anodeMainPnP2AxisZ.monitoring.busy;
   "Unit1.EmNodes".allBrakeTest.monitoring.emStatus.complete[12] := "Unit1.Em4.ControlNodes".cm.brakeTest.anodeMainPnP1AxisZ.monitoring.complete;
   "Unit1.EmNodes".allBrakeTest.monitoring.emStatus.complete[14] := "Unit1.Em4.ControlNodes".cm.brakeTest.anodeMainPnP2AxisZ.monitoring.complete;
   "Unit1.EmNodes".allBrakeTest.monitoring.emStatus.axisEnabled[12] := "Unit1.Em4.ControlNodes".cm.brakeTest.anodeMainPnP1AxisZ.monitoring.ready;
   "Unit1.EmNodes".allBrakeTest.monitoring.emStatus.axisEnabled[14] := "Unit1.Em4.ControlNodes".cm.brakeTest.anodeMainPnP2AxisZ.monitoring.ready;
END_REGION

REGION Network 305: Em Relations Home Check
   RUNG wire#powerrail
      Move(in := "Unit1.Em4.ControlNodes".mainPnP.preOperationCheck, out1 => "Unit1.EmNodes".emRelations.em04.sequence.Spare1.preOperationCheck)
      Move(in := "Unit1.Em4.ControlNodes".alignTable.preOperationCheck, out1 => "Unit1.EmNodes".emRelations.em04.sequence.Spare2.preOperationCheck)
      Move(in := "Unit1.Em4.ControlNodes".ngPnP.preOperationCheck, out1 => "Unit1.EmNodes".emRelations.em04.sequence.Spare3.preOperationCheck)
   END_RUNG
   // the same network as SCL:
   "Unit1.EmNodes".emRelations.em04.sequence.Spare1.preOperationCheck := "Unit1.Em4.ControlNodes".mainPnP.preOperationCheck;
   "Unit1.EmNodes".emRelations.em04.sequence.Spare2.preOperationCheck := "Unit1.Em4.ControlNodes".alignTable.preOperationCheck;
   "Unit1.EmNodes".emRelations.em04.sequence.Spare3.preOperationCheck := "Unit1.Em4.ControlNodes".ngPnP.preOperationCheck;
END_REGION

REGION Network 306: Em Relations Cylinder
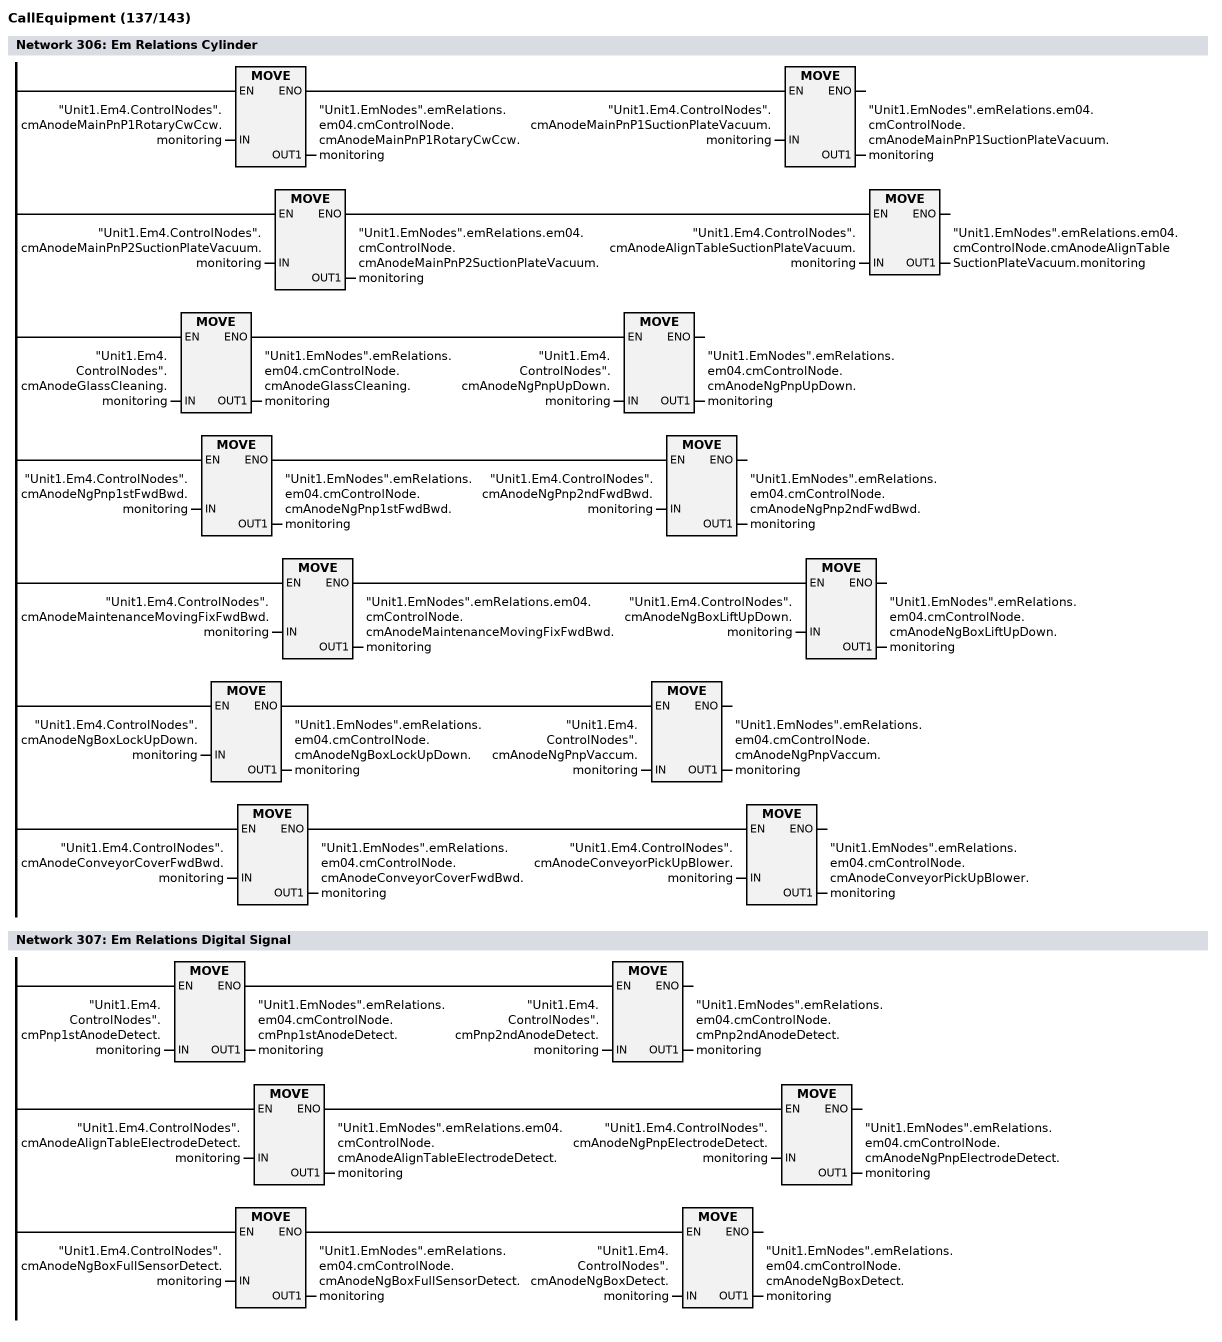
   RUNG wire#powerrail
      Move(in := "Unit1.Em4.ControlNodes".cmAnodeMainPnP1RotaryCwCcw.monitoring, out1 => "Unit1.EmNodes".emRelations.em04.cmControlNode.cmAnodeMainPnP1RotaryCwCcw.monitoring)
      Move(in := "Unit1.Em4.ControlNodes".cmAnodeMainPnP1SuctionPlateVacuum.monitoring, out1 => "Unit1.EmNodes".emRelations.em04.cmControlNode.cmAnodeMainPnP1SuctionPlateVacuum.monitoring)
   END_RUNG
   RUNG wire#powerrail
      Move(in := "Unit1.Em4.ControlNodes".cmAnodeMainPnP2SuctionPlateVacuum.monitoring, out1 => "Unit1.EmNodes".emRelations.em04.cmControlNode.cmAnodeMainPnP2SuctionPlateVacuum.monitoring)
      Move(in := "Unit1.Em4.ControlNodes".cmAnodeAlignTableSuctionPlateVacuum.monitoring, out1 => "Unit1.EmNodes".emRelations.em04.cmControlNode.cmAnodeAlignTableSuctionPlateVacuum.monitoring)
   END_RUNG
   RUNG wire#powerrail
      Move(in := "Unit1.Em4.ControlNodes".cmAnodeGlassCleaning.monitoring, out1 => "Unit1.EmNodes".emRelations.em04.cmControlNode.cmAnodeGlassCleaning.monitoring)
      Move(in := "Unit1.Em4.ControlNodes".cmAnodeNgPnpUpDown.monitoring, out1 => "Unit1.EmNodes".emRelations.em04.cmControlNode.cmAnodeNgPnpUpDown.monitoring)
   END_RUNG
   RUNG wire#powerrail
      Move(in := "Unit1.Em4.ControlNodes".cmAnodeNgPnp1stFwdBwd.monitoring, out1 => "Unit1.EmNodes".emRelations.em04.cmControlNode.cmAnodeNgPnp1stFwdBwd.monitoring)
      Move(in := "Unit1.Em4.ControlNodes".cmAnodeNgPnp2ndFwdBwd.monitoring, out1 => "Unit1.EmNodes".emRelations.em04.cmControlNode.cmAnodeNgPnp2ndFwdBwd.monitoring)
   END_RUNG
   RUNG wire#powerrail
      Move(in := "Unit1.Em4.ControlNodes".cmAnodeMaintenanceMovingFixFwdBwd.monitoring, out1 => "Unit1.EmNodes".emRelations.em04.cmControlNode.cmAnodeMaintenanceMovingFixFwdBwd.monitoring)
      Move(in := "Unit1.Em4.ControlNodes".cmAnodeNgBoxLiftUpDown.monitoring, out1 => "Unit1.EmNodes".emRelations.em04.cmControlNode.cmAnodeNgBoxLiftUpDown.monitoring)
   END_RUNG
   RUNG wire#powerrail
      Move(in := "Unit1.Em4.ControlNodes".cmAnodeNgBoxLockUpDown.monitoring, out1 => "Unit1.EmNodes".emRelations.em04.cmControlNode.cmAnodeNgBoxLockUpDown.monitoring)
      Move(in := "Unit1.Em4.ControlNodes".cmAnodeNgPnpVaccum.monitoring, out1 => "Unit1.EmNodes".emRelations.em04.cmControlNode.cmAnodeNgPnpVaccum.monitoring)
   END_RUNG
   RUNG wire#powerrail
      Move(in := "Unit1.Em4.ControlNodes".cmAnodeConveyorCoverFwdBwd.monitoring, out1 => "Unit1.EmNodes".emRelations.em04.cmControlNode.cmAnodeConveyorCoverFwdBwd.monitoring)
      Move(in := "Unit1.Em4.ControlNodes".cmAnodeConveyorPickUpBlower.monitoring, out1 => "Unit1.EmNodes".emRelations.em04.cmControlNode.cmAnodeConveyorPickUpBlower.monitoring)
   END_RUNG
   // the same network as SCL:
   "Unit1.EmNodes".emRelations.em04.cmControlNode.cmAnodeMainPnP1RotaryCwCcw.monitoring := "Unit1.Em4.ControlNodes".cmAnodeMainPnP1RotaryCwCcw.monitoring;
   "Unit1.EmNodes".emRelations.em04.cmControlNode.cmAnodeMainPnP1SuctionPlateVacuum.monitoring := "Unit1.Em4.ControlNodes".cmAnodeMainPnP1SuctionPlateVacuum.monitoring;
   "Unit1.EmNodes".emRelations.em04.cmControlNode.cmAnodeMainPnP2SuctionPlateVacuum.monitoring := "Unit1.Em4.ControlNodes".cmAnodeMainPnP2SuctionPlateVacuum.monitoring;
   "Unit1.EmNodes".emRelations.em04.cmControlNode.cmAnodeAlignTableSuctionPlateVacuum.monitoring := "Unit1.Em4.ControlNodes".cmAnodeAlignTableSuctionPlateVacuum.monitoring;
   "Unit1.EmNodes".emRelations.em04.cmControlNode.cmAnodeGlassCleaning.monitoring := "Unit1.Em4.ControlNodes".cmAnodeGlassCleaning.monitoring;
   "Unit1.EmNodes".emRelations.em04.cmControlNode.cmAnodeNgPnpUpDown.monitoring := "Unit1.Em4.ControlNodes".cmAnodeNgPnpUpDown.monitoring;
   "Unit1.EmNodes".emRelations.em04.cmControlNode.cmAnodeNgPnp1stFwdBwd.monitoring := "Unit1.Em4.ControlNodes".cmAnodeNgPnp1stFwdBwd.monitoring;
   "Unit1.EmNodes".emRelations.em04.cmControlNode.cmAnodeNgPnp2ndFwdBwd.monitoring := "Unit1.Em4.ControlNodes".cmAnodeNgPnp2ndFwdBwd.monitoring;
   "Unit1.EmNodes".emRelations.em04.cmControlNode.cmAnodeMaintenanceMovingFixFwdBwd.monitoring := "Unit1.Em4.ControlNodes".cmAnodeMaintenanceMovingFixFwdBwd.monitoring;
   "Unit1.EmNodes".emRelations.em04.cmControlNode.cmAnodeNgBoxLiftUpDown.monitoring := "Unit1.Em4.ControlNodes".cmAnodeNgBoxLiftUpDown.monitoring;
   "Unit1.EmNodes".emRelations.em04.cmControlNode.cmAnodeNgBoxLockUpDown.monitoring := "Unit1.Em4.ControlNodes".cmAnodeNgBoxLockUpDown.monitoring;
   "Unit1.EmNodes".emRelations.em04.cmControlNode.cmAnodeNgPnpVaccum.monitoring := "Unit1.Em4.ControlNodes".cmAnodeNgPnpVaccum.monitoring;
   "Unit1.EmNodes".emRelations.em04.cmControlNode.cmAnodeConveyorCoverFwdBwd.monitoring := "Unit1.Em4.ControlNodes".cmAnodeConveyorCoverFwdBwd.monitoring;
   "Unit1.EmNodes".emRelations.em04.cmControlNode.cmAnodeConveyorPickUpBlower.monitoring := "Unit1.Em4.ControlNodes".cmAnodeConveyorPickUpBlower.monitoring;
END_REGION

REGION Network 307: Em Relations Digital Signal
   RUNG wire#powerrail
      Move(in := "Unit1.Em4.ControlNodes".cmPnp1stAnodeDetect.monitoring, out1 => "Unit1.EmNodes".emRelations.em04.cmControlNode.cmPnp1stAnodeDetect.monitoring)
      Move(in := "Unit1.Em4.ControlNodes".cmPnp2ndAnodeDetect.monitoring, out1 => "Unit1.EmNodes".emRelations.em04.cmControlNode.cmPnp2ndAnodeDetect.monitoring)
   END_RUNG
   RUNG wire#powerrail
      Move(in := "Unit1.Em4.ControlNodes".cmAnodeAlignTableElectrodeDetect.monitoring, out1 => "Unit1.EmNodes".emRelations.em04.cmControlNode.cmAnodeAlignTableElectrodeDetect.monitoring)
      Move(in := "Unit1.Em4.ControlNodes".cmAnodeNgPnpElectrodeDetect.monitoring, out1 => "Unit1.EmNodes".emRelations.em04.cmControlNode.cmAnodeNgPnpElectrodeDetect.monitoring)
   END_RUNG
   RUNG wire#powerrail
      Move(in := "Unit1.Em4.ControlNodes".cmAnodeNgBoxFullSensorDetect.monitoring, out1 => "Unit1.EmNodes".emRelations.em04.cmControlNode.cmAnodeNgBoxFullSensorDetect.monitoring)
      Move(in := "Unit1.Em4.ControlNodes".cmAnodeNgBoxDetect.monitoring, out1 => "Unit1.EmNodes".emRelations.em04.cmControlNode.cmAnodeNgBoxDetect.monitoring)
   END_RUNG
   // the same network as SCL:
   "Unit1.EmNodes".emRelations.em04.cmControlNode.cmPnp1stAnodeDetect.monitoring := "Unit1.Em4.ControlNodes".cmPnp1stAnodeDetect.monitoring;
   "Unit1.EmNodes".emRelations.em04.cmControlNode.cmPnp2ndAnodeDetect.monitoring := "Unit1.Em4.ControlNodes".cmPnp2ndAnodeDetect.monitoring;
   "Unit1.EmNodes".emRelations.em04.cmControlNode.cmAnodeAlignTableElectrodeDetect.monitoring := "Unit1.Em4.ControlNodes".cmAnodeAlignTableElectrodeDetect.monitoring;
   "Unit1.EmNodes".emRelations.em04.cmControlNode.cmAnodeNgPnpElectrodeDetect.monitoring := "Unit1.Em4.ControlNodes".cmAnodeNgPnpElectrodeDetect.monitoring;
   "Unit1.EmNodes".emRelations.em04.cmControlNode.cmAnodeNgBoxFullSensorDetect.monitoring := "Unit1.Em4.ControlNodes".cmAnodeNgBoxFullSensorDetect.monitoring;
   "Unit1.EmNodes".emRelations.em04.cmControlNode.cmAnodeNgBoxDetect.monitoring := "Unit1.Em4.ControlNodes".cmAnodeNgBoxDetect.monitoring;
END_REGION

REGION Network 308: Em Relations Sequence Interface
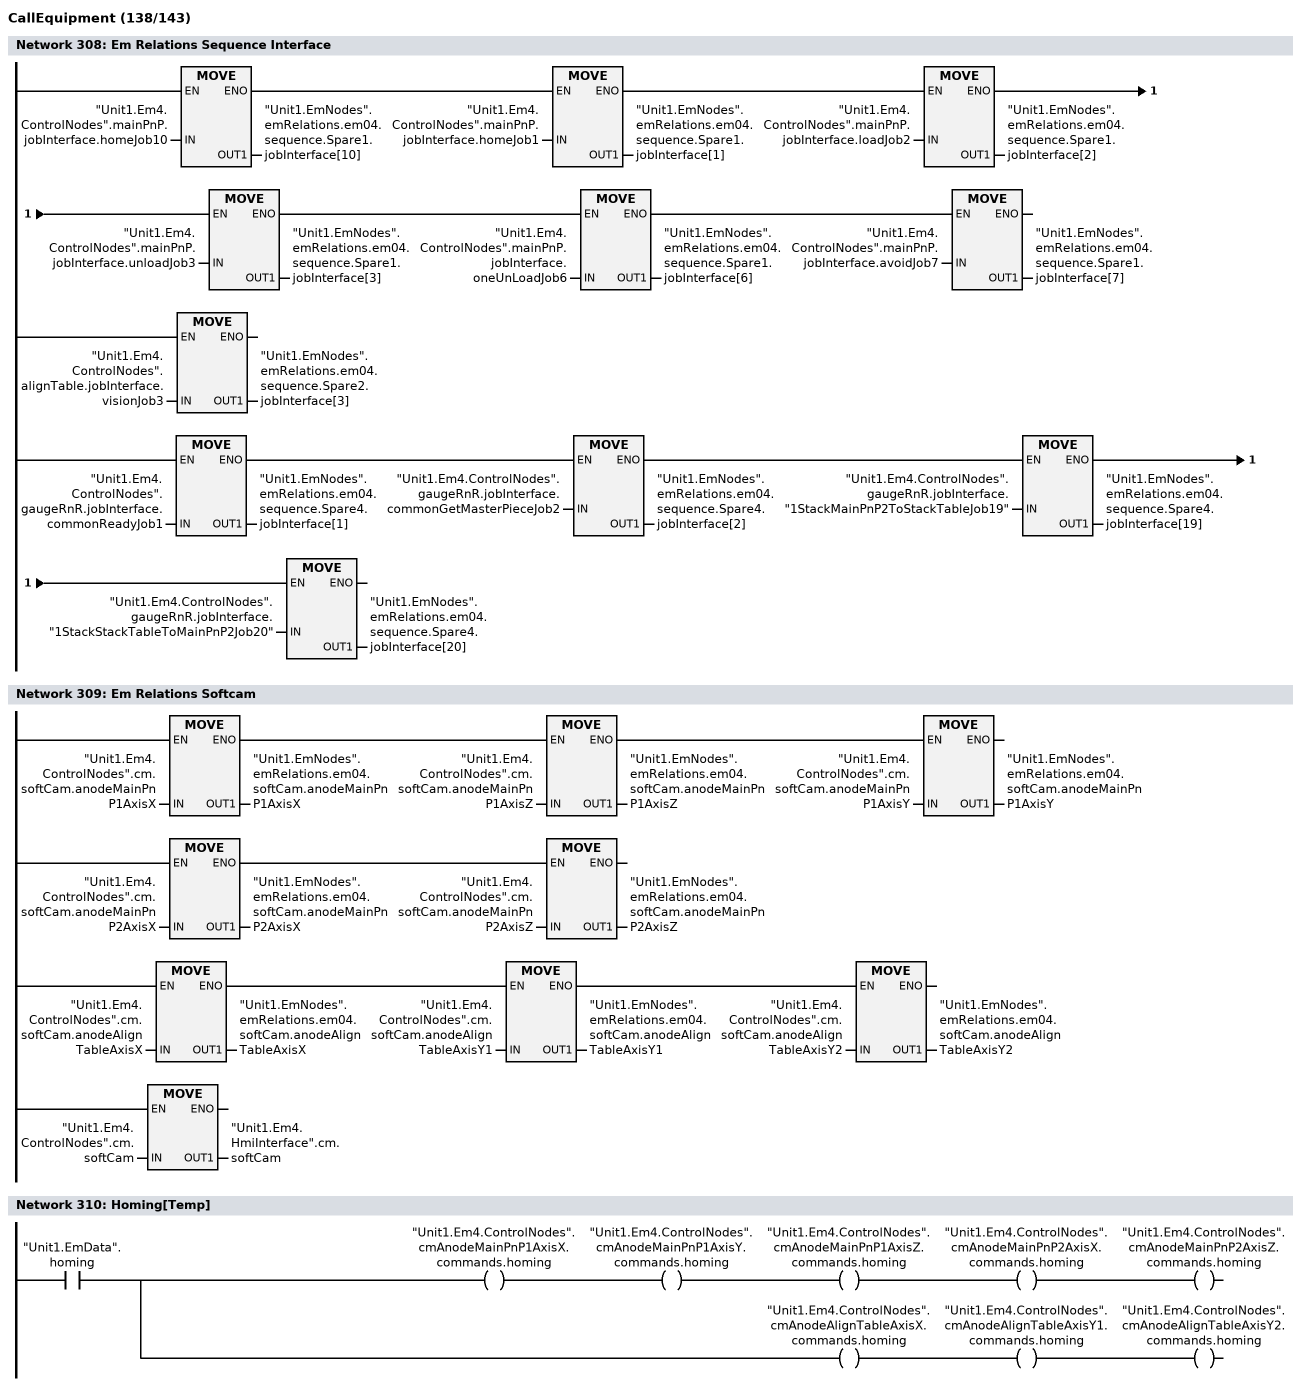
   RUNG wire#powerrail
      Move(in := "Unit1.Em4.ControlNodes".mainPnP.jobInterface.homeJob10, out1 => "Unit1.EmNodes".emRelations.em04.sequence.Spare1.jobInterface[10])
      Move(in := "Unit1.Em4.ControlNodes".mainPnP.jobInterface.homeJob1, out1 => "Unit1.EmNodes".emRelations.em04.sequence.Spare1.jobInterface[1])
      Move(in := "Unit1.Em4.ControlNodes".mainPnP.jobInterface.loadJob2, out1 => "Unit1.EmNodes".emRelations.em04.sequence.Spare1.jobInterface[2])
      Move(in := "Unit1.Em4.ControlNodes".mainPnP.jobInterface.unloadJob3, out1 => "Unit1.EmNodes".emRelations.em04.sequence.Spare1.jobInterface[3])
      Move(in := "Unit1.Em4.ControlNodes".mainPnP.jobInterface.oneUnLoadJob6, out1 => "Unit1.EmNodes".emRelations.em04.sequence.Spare1.jobInterface[6])
      Move(in := "Unit1.Em4.ControlNodes".mainPnP.jobInterface.avoidJob7, out1 => "Unit1.EmNodes".emRelations.em04.sequence.Spare1.jobInterface[7])
   END_RUNG
   RUNG wire#powerrail
      Move(in := "Unit1.Em4.ControlNodes".alignTable.jobInterface.visionJob3, out1 => "Unit1.EmNodes".emRelations.em04.sequence.Spare2.jobInterface[3])
   END_RUNG
   RUNG wire#powerrail
      Move(in := "Unit1.Em4.ControlNodes".gaugeRnR.jobInterface.commonReadyJob1, out1 => "Unit1.EmNodes".emRelations.em04.sequence.Spare4.jobInterface[1])
      Move(in := "Unit1.Em4.ControlNodes".gaugeRnR.jobInterface.commonGetMasterPieceJob2, out1 => "Unit1.EmNodes".emRelations.em04.sequence.Spare4.jobInterface[2])
      Move(in := "Unit1.Em4.ControlNodes".gaugeRnR.jobInterface."1StackMainPnP2ToStackTableJob19", out1 => "Unit1.EmNodes".emRelations.em04.sequence.Spare4.jobInterface[19])
      Move(in := "Unit1.Em4.ControlNodes".gaugeRnR.jobInterface."1StackStackTableToMainPnP2Job20", out1 => "Unit1.EmNodes".emRelations.em04.sequence.Spare4.jobInterface[20])
   END_RUNG
   // the same network as SCL:
   "Unit1.EmNodes".emRelations.em04.sequence.Spare1.jobInterface[10] := "Unit1.Em4.ControlNodes".mainPnP.jobInterface.homeJob10;
   "Unit1.EmNodes".emRelations.em04.sequence.Spare1.jobInterface[1] := "Unit1.Em4.ControlNodes".mainPnP.jobInterface.homeJob1;
   "Unit1.EmNodes".emRelations.em04.sequence.Spare1.jobInterface[2] := "Unit1.Em4.ControlNodes".mainPnP.jobInterface.loadJob2;
   "Unit1.EmNodes".emRelations.em04.sequence.Spare1.jobInterface[3] := "Unit1.Em4.ControlNodes".mainPnP.jobInterface.unloadJob3;
   "Unit1.EmNodes".emRelations.em04.sequence.Spare1.jobInterface[6] := "Unit1.Em4.ControlNodes".mainPnP.jobInterface.oneUnLoadJob6;
   "Unit1.EmNodes".emRelations.em04.sequence.Spare1.jobInterface[7] := "Unit1.Em4.ControlNodes".mainPnP.jobInterface.avoidJob7;
   "Unit1.EmNodes".emRelations.em04.sequence.Spare2.jobInterface[3] := "Unit1.Em4.ControlNodes".alignTable.jobInterface.visionJob3;
   "Unit1.EmNodes".emRelations.em04.sequence.Spare4.jobInterface[1] := "Unit1.Em4.ControlNodes".gaugeRnR.jobInterface.commonReadyJob1;
   "Unit1.EmNodes".emRelations.em04.sequence.Spare4.jobInterface[2] := "Unit1.Em4.ControlNodes".gaugeRnR.jobInterface.commonGetMasterPieceJob2;
   "Unit1.EmNodes".emRelations.em04.sequence.Spare4.jobInterface[19] := "Unit1.Em4.ControlNodes".gaugeRnR.jobInterface."1StackMainPnP2ToStackTableJob19";
   "Unit1.EmNodes".emRelations.em04.sequence.Spare4.jobInterface[20] := "Unit1.Em4.ControlNodes".gaugeRnR.jobInterface."1StackStackTableToMainPnP2Job20";
END_REGION

REGION Network 309: Em Relations Softcam
   RUNG wire#powerrail
      Move(in := "Unit1.Em4.ControlNodes".cm.softCam.anodeMainPnP1AxisX, out1 => "Unit1.EmNodes".emRelations.em04.softCam.anodeMainPnP1AxisX)
      Move(in := "Unit1.Em4.ControlNodes".cm.softCam.anodeMainPnP1AxisZ, out1 => "Unit1.EmNodes".emRelations.em04.softCam.anodeMainPnP1AxisZ)
      Move(in := "Unit1.Em4.ControlNodes".cm.softCam.anodeMainPnP1AxisY, out1 => "Unit1.EmNodes".emRelations.em04.softCam.anodeMainPnP1AxisY)
   END_RUNG
   RUNG wire#powerrail
      Move(in := "Unit1.Em4.ControlNodes".cm.softCam.anodeMainPnP2AxisX, out1 => "Unit1.EmNodes".emRelations.em04.softCam.anodeMainPnP2AxisX)
      Move(in := "Unit1.Em4.ControlNodes".cm.softCam.anodeMainPnP2AxisZ, out1 => "Unit1.EmNodes".emRelations.em04.softCam.anodeMainPnP2AxisZ)
   END_RUNG
   RUNG wire#powerrail
      Move(in := "Unit1.Em4.ControlNodes".cm.softCam.anodeAlignTableAxisX, out1 => "Unit1.EmNodes".emRelations.em04.softCam.anodeAlignTableAxisX)
      Move(in := "Unit1.Em4.ControlNodes".cm.softCam.anodeAlignTableAxisY1, out1 => "Unit1.EmNodes".emRelations.em04.softCam.anodeAlignTableAxisY1)
      Move(in := "Unit1.Em4.ControlNodes".cm.softCam.anodeAlignTableAxisY2, out1 => "Unit1.EmNodes".emRelations.em04.softCam.anodeAlignTableAxisY2)
   END_RUNG
   RUNG wire#powerrail
      Move(in := "Unit1.Em4.ControlNodes".cm.softCam, out1 => "Unit1.Em4.HmiInterface".cm.softCam)
   END_RUNG
   // the same network as SCL:
   "Unit1.EmNodes".emRelations.em04.softCam.anodeMainPnP1AxisX := "Unit1.Em4.ControlNodes".cm.softCam.anodeMainPnP1AxisX;
   "Unit1.EmNodes".emRelations.em04.softCam.anodeMainPnP1AxisZ := "Unit1.Em4.ControlNodes".cm.softCam.anodeMainPnP1AxisZ;
   "Unit1.EmNodes".emRelations.em04.softCam.anodeMainPnP1AxisY := "Unit1.Em4.ControlNodes".cm.softCam.anodeMainPnP1AxisY;
   "Unit1.EmNodes".emRelations.em04.softCam.anodeMainPnP2AxisX := "Unit1.Em4.ControlNodes".cm.softCam.anodeMainPnP2AxisX;
   "Unit1.EmNodes".emRelations.em04.softCam.anodeMainPnP2AxisZ := "Unit1.Em4.ControlNodes".cm.softCam.anodeMainPnP2AxisZ;
   "Unit1.EmNodes".emRelations.em04.softCam.anodeAlignTableAxisX := "Unit1.Em4.ControlNodes".cm.softCam.anodeAlignTableAxisX;
   "Unit1.EmNodes".emRelations.em04.softCam.anodeAlignTableAxisY1 := "Unit1.Em4.ControlNodes".cm.softCam.anodeAlignTableAxisY1;
   "Unit1.EmNodes".emRelations.em04.softCam.anodeAlignTableAxisY2 := "Unit1.Em4.ControlNodes".cm.softCam.anodeAlignTableAxisY2;
   "Unit1.Em4.HmiInterface".cm.softCam := "Unit1.Em4.ControlNodes".cm.softCam;
END_REGION

REGION Network 310: Homing[Temp]
   RUNG wire#powerrail
      Contact( "Unit1.EmData".homing )
      wire#w1
      Coil( "Unit1.Em4.ControlNodes".cmAnodeMainPnP1AxisX.commands.homing )
      Coil( "Unit1.Em4.ControlNodes".cmAnodeMainPnP1AxisY.commands.homing )
      Coil( "Unit1.Em4.ControlNodes".cmAnodeMainPnP1AxisZ.commands.homing )
      Coil( "Unit1.Em4.ControlNodes".cmAnodeMainPnP2AxisX.commands.homing )
      Coil( "Unit1.Em4.ControlNodes".cmAnodeMainPnP2AxisZ.commands.homing )
   END_RUNG
   RUNG wire#w1
      Coil( "Unit1.Em4.ControlNodes".cmAnodeAlignTableAxisX.commands.homing )
      Coil( "Unit1.Em4.ControlNodes".cmAnodeAlignTableAxisY1.commands.homing )
      Coil( "Unit1.Em4.ControlNodes".cmAnodeAlignTableAxisY2.commands.homing )
   END_RUNG
   // the same network as SCL:
   "Unit1.Em4.ControlNodes".cmAnodeMainPnP1AxisX.commands.homing := "Unit1.EmData".homing;
   "Unit1.Em4.ControlNodes".cmAnodeMainPnP1AxisY.commands.homing := "Unit1.EmData".homing;
   "Unit1.Em4.ControlNodes".cmAnodeMainPnP1AxisZ.commands.homing := "Unit1.EmData".homing;
   "Unit1.Em4.ControlNodes".cmAnodeMainPnP2AxisX.commands.homing := "Unit1.EmData".homing;
   "Unit1.Em4.ControlNodes".cmAnodeMainPnP2AxisZ.commands.homing := "Unit1.EmData".homing;
   "Unit1.Em4.ControlNodes".cmAnodeAlignTableAxisX.commands.homing := "Unit1.EmData".homing;
   "Unit1.Em4.ControlNodes".cmAnodeAlignTableAxisY1.commands.homing := "Unit1.EmData".homing;
   "Unit1.Em4.ControlNodes".cmAnodeAlignTableAxisY2.commands.homing := "Unit1.EmData".homing;
END_REGION

REGION Network 311
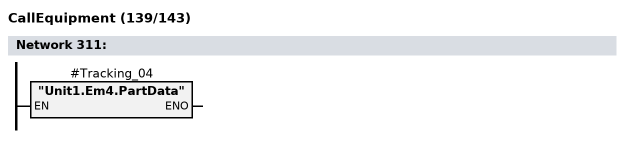
   RUNG wire#powerrail
      #Tracking_04()
   END_RUNG
   // the same network as SCL:
   #Tracking_04();   // "Unit1.Em4.PartData"
END_REGION

REGION Network 312 (SCL): SyncMotion Configuration
   "Unit1.MotionNodes".PLCToMotion.TechnologyObject.Axis.AnodePnPX1 := "Unit1.Em4.Config".axis[1];
   "Unit1.MotionNodes".PLCToMotion.TechnologyObject.Axis.AnodePnPX2 := "Unit1.Em4.Config".axis[2];
   "Unit1.MotionNodes".PLCToMotion.TechnologyObject.Axis.AnodePnPZ1 := "Unit1.Em4.Config".axis[4];
   "Unit1.MotionNodes".PLCToMotion.TechnologyObject.Axis.AnodePnPZ2 := "Unit1.Em4.Config".axis[5];


   // _.Unit1.SyncMotion.Configuration.TechnologyObjects.StackMain.Cam.AnodePnPX1Cam := Config.cam[1];
   // _.Unit1.SyncMotion.Configuration.TechnologyObjects.StackMain.Cam.AnodePnPX2Cam := Config.cam[2];
   // _.Unit1.SyncMotion.Configuration.TechnologyObjects.StackMain.Cam.AnodePnPZ1Cam := Config.cam[3];
   // _.Unit1.SyncMotion.Configuration.TechnologyObjects.StackMain.Cam.AnodePnPZ2Cam := Config.cam[4];

   "Unit1.Em4.Config".outputCam[1] := "AnodePnP1XFwd";
   "Unit1.Em4.Config".outputCam[2] := "AnodePnP1XBwd";
   "Unit1.Em4.Config".outputCam[3] := "AnodePnP2XFwd";
   "Unit1.Em4.Config".outputCam[4] := "AnodePnP2XBwd";
   "Unit1.Em4.Config".outputCam[5] := "AnodePnPZ1Down1";
   "Unit1.Em4.Config".outputCam[6] := "AnodePnPZ1Up1";
   "Unit1.Em4.Config".outputCam[7] := "AnodePnPZ2Down1";
   "Unit1.Em4.Config".outputCam[8] := "AnodePnPZ2Up1";
   "Unit1.Em4.Config".outputCam[9] := "AnodePnPZ1Down2";
   "Unit1.Em4.Config".outputCam[10] := "AnodePnPZ1Up2";
   "Unit1.Em4.Config".outputCam[11] := "AnodePnPZ2Down2";
   "Unit1.Em4.Config".outputCam[12] := "AnodePnPZ2Up2";
   "Unit1.Em4.Config".outputCam[13] := "AnodePnPZ1SuctionOn";
   "Unit1.Em4.Config".outputCam[14] := "AnodePnPZ1SuctionOff";
   "Unit1.Em4.Config".outputCam[15] := "AnodePnPZ1ReelCutBlow";
   "Unit1.Em4.Config".outputCam[16] := "AnodePnPZ2SuctionOn";
   "Unit1.Em4.Config".outputCam[17] := "AnodePnPZ2SuctionOff";
   "Unit1.Em4.Config".outputCam[18] := "AnodeAlignSuctionOn";
   "Unit1.Em4.Config".outputCam[19] := "AnodeAlignSuctionOff";
   "Unit1.Em4.Config".outputCam[20] := "AnodePnPZ1ReelCutDataDeleteOn";
   "Unit1.Em4.Config".outputCam[21] := "AnodePnP1XReelCutDataDeleteOff";
   "Unit1.Em4.Config".outputCam[22] := "AnodeAlignVision";

   "Unit1.MotionNodes".PLCToMotion.TechnologyObject.OutputCam.AnodePnPX1BwdOutputCam := "Unit1.Em4.Config".outputCam[1];
   "Unit1.MotionNodes".PLCToMotion.TechnologyObject.OutputCam.AnodePnPX1FwdOutputCam := "Unit1.Em4.Config".outputCam[2];
   "Unit1.MotionNodes".PLCToMotion.TechnologyObject.OutputCam.AnodePnPX2BwdOutputCam := "Unit1.Em4.Config".outputCam[3];
   "Unit1.MotionNodes".PLCToMotion.TechnologyObject.OutputCam.AnodePnPX2FwdOutputCam := "Unit1.Em4.Config".outputCam[4];
   "Unit1.MotionNodes".PLCToMotion.TechnologyObject.OutputCam.AnodePnPZ1Down1OutputCam := "Unit1.Em4.Config".outputCam[5];
   "Unit1.MotionNodes".PLCToMotion.TechnologyObject.OutputCam.AnodePnPZ1Up1OutputCam := "Unit1.Em4.Config".outputCam[6];
   "Unit1.MotionNodes".PLCToMotion.TechnologyObject.OutputCam.AnodePnPZ2Down1OutputCam := "Unit1.Em4.Config".outputCam[7];
   "Unit1.MotionNodes".PLCToMotion.TechnologyObject.OutputCam.AnodePnPZ2Up1OutputCam := "Unit1.Em4.Config".outputCam[8];
   "Unit1.MotionNodes".PLCToMotion.TechnologyObject.OutputCam.AnodePnPZ1Down2OutputCam := "Unit1.Em4.Config".outputCam[9];
   "Unit1.MotionNodes".PLCToMotion.TechnologyObject.OutputCam.AnodePnPZ1Up2OutputCam := "Unit1.Em4.Config".outputCam[10];
   "Unit1.MotionNodes".PLCToMotion.TechnologyObject.OutputCam.AnodePnPZ2Down2OutputCam := "Unit1.Em4.Config".outputCam[11];
   "Unit1.MotionNodes".PLCToMotion.TechnologyObject.OutputCam.AnodePnPZ2Up2OutputCam := "Unit1.Em4.Config".outputCam[12];
   "Unit1.MotionNodes".PLCToMotion.TechnologyObject.OutputCam.AnodePnPZ1SuctionOnOutputCam := "Unit1.Em4.Config".outputCam[13];
   "Unit1.MotionNodes".PLCToMotion.TechnologyObject.OutputCam.AnodePnPZ1SuctionOffOutputCam := "Unit1.Em4.Config".outputCam[14];
   "Unit1.MotionNodes".PLCToMotion.TechnologyObject.OutputCam.AnodePnPZ1ReelCutBlowOutputCam := "Unit1.Em4.Config".outputCam[15];
   "Unit1.MotionNodes".PLCToMotion.TechnologyObject.OutputCam.AnodePnPZ2SuctionOnOutputCam := "Unit1.Em4.Config".outputCam[16];
   "Unit1.MotionNodes".PLCToMotion.TechnologyObject.OutputCam.AnodePnPZ2SuctionOffOutputCam := "Unit1.Em4.Config".outputCam[17];
   "Unit1.MotionNodes".PLCToMotion.TechnologyObject.OutputCam.AnodeAlignSuctionOnOutputCam := "Unit1.Em4.Config".outputCam[18];
   "Unit1.MotionNodes".PLCToMotion.TechnologyObject.OutputCam.AnodeAlignSuctionOffOutputCam := "Unit1.Em4.Config".outputCam[19];
   "Unit1.MotionNodes".PLCToMotion.TechnologyObject.OutputCam.AnodePnPZ1ReelCutDataDeleteOnOutputCam := "Unit1.Em4.Config".outputCam[20];
   "Unit1.MotionNodes".PLCToMotion.TechnologyObject.OutputCam.AnodePnP1XReelCutDataDeleteOffOutputCam := "Unit1.Em4.Config".outputCam[21];
   "Unit1.MotionNodes".PLCToMotion.TechnologyObject.OutputCam.AnodeAlignVisionOutputCam := "Unit1.Em4.Config".outputCam[22];
END_REGION

REGION Network 313: Axis
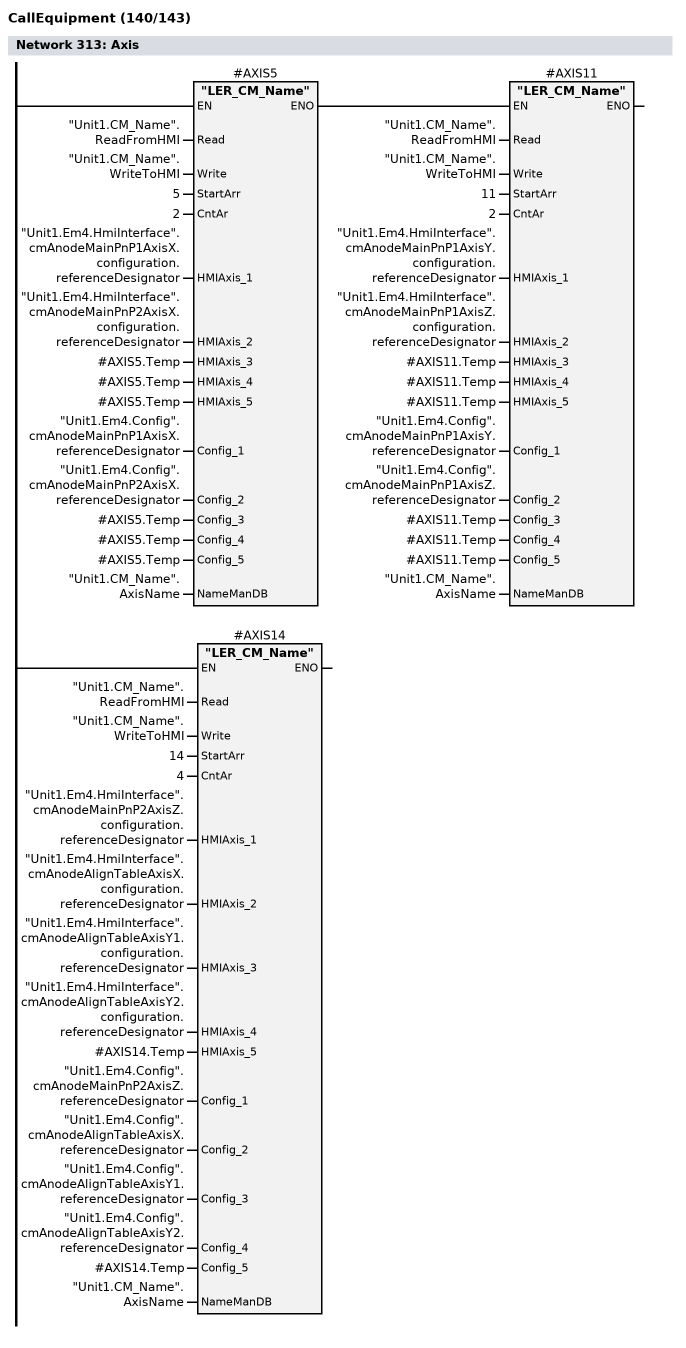
   RUNG wire#powerrail
      #AXIS5(Read := "Unit1.CM_Name".ReadFromHMI, Write := "Unit1.CM_Name".WriteToHMI, StartArr := 5, CntAr := 2, HMIAxis_1 := "Unit1.Em4.HmiInterface".cmAnodeMainPnP1AxisX.configuration.referenceDesignator, HMIAxis_2 := "Unit1.Em4.HmiInterface".cmAnodeMainPnP2AxisX.configuration.referenceDesignator, HMIAxis_3 := #AXIS5.Temp, HMIAxis_4 := #AXIS5.Temp, HMIAxis_5 := #AXIS5.Temp, Config_1 := "Unit1.Em4.Config".cmAnodeMainPnP1AxisX.referenceDesignator, Config_2 := "Unit1.Em4.Config".cmAnodeMainPnP2AxisX.referenceDesignator, Config_3 := #AXIS5.Temp, Config_4 := #AXIS5.Temp, Config_5 := #AXIS5.Temp, NameManDB := "Unit1.CM_Name".AxisName)
      #AXIS11(Read := "Unit1.CM_Name".ReadFromHMI, Write := "Unit1.CM_Name".WriteToHMI, StartArr := 11, CntAr := 2, HMIAxis_1 := "Unit1.Em4.HmiInterface".cmAnodeMainPnP1AxisY.configuration.referenceDesignator, HMIAxis_2 := "Unit1.Em4.HmiInterface".cmAnodeMainPnP1AxisZ.configuration.referenceDesignator, HMIAxis_3 := #AXIS11.Temp, HMIAxis_4 := #AXIS11.Temp, HMIAxis_5 := #AXIS11.Temp, Config_1 := "Unit1.Em4.Config".cmAnodeMainPnP1AxisY.referenceDesignator, Config_2 := "Unit1.Em4.Config".cmAnodeMainPnP1AxisZ.referenceDesignator, Config_3 := #AXIS11.Temp, Config_4 := #AXIS11.Temp, Config_5 := #AXIS11.Temp, NameManDB := "Unit1.CM_Name".AxisName)
   END_RUNG
   RUNG wire#powerrail
      #AXIS14(Read := "Unit1.CM_Name".ReadFromHMI, Write := "Unit1.CM_Name".WriteToHMI, StartArr := 14, CntAr := 4, HMIAxis_1 := "Unit1.Em4.HmiInterface".cmAnodeMainPnP2AxisZ.configuration.referenceDesignator, HMIAxis_2 := "Unit1.Em4.HmiInterface".cmAnodeAlignTableAxisX.configuration.referenceDesignator, HMIAxis_3 := "Unit1.Em4.HmiInterface".cmAnodeAlignTableAxisY1.configuration.referenceDesignator, HMIAxis_4 := "Unit1.Em4.HmiInterface".cmAnodeAlignTableAxisY2.configuration.referenceDesignator, HMIAxis_5 := #AXIS14.Temp, Config_1 := "Unit1.Em4.Config".cmAnodeMainPnP2AxisZ.referenceDesignator, Config_2 := "Unit1.Em4.Config".cmAnodeAlignTableAxisX.referenceDesignator, Config_3 := "Unit1.Em4.Config".cmAnodeAlignTableAxisY1.referenceDesignator, Config_4 := "Unit1.Em4.Config".cmAnodeAlignTableAxisY2.referenceDesignator, Config_5 := #AXIS14.Temp, NameManDB := "Unit1.CM_Name".AxisName)
   END_RUNG
   // the same network as SCL:
   #AXIS5(Read := "Unit1.CM_Name".ReadFromHMI,   // "LER_CM_Name"
          Write := "Unit1.CM_Name".WriteToHMI,
          StartArr := 5,
          CntAr := 2,
          HMIAxis_1 := "Unit1.Em4.HmiInterface".cmAnodeMainPnP1AxisX.configuration.referenceDesignator,
          HMIAxis_2 := "Unit1.Em4.HmiInterface".cmAnodeMainPnP2AxisX.configuration.referenceDesignator,
          HMIAxis_3 := #AXIS5.Temp,
          HMIAxis_4 := #AXIS5.Temp,
          HMIAxis_5 := #AXIS5.Temp,
          Config_1 := "Unit1.Em4.Config".cmAnodeMainPnP1AxisX.referenceDesignator,
          Config_2 := "Unit1.Em4.Config".cmAnodeMainPnP2AxisX.referenceDesignator,
          Config_3 := #AXIS5.Temp,
          Config_4 := #AXIS5.Temp,
          Config_5 := #AXIS5.Temp,
          NameManDB := "Unit1.CM_Name".AxisName,
          ENO => #_w1);
   IF #_w1 THEN
       #AXIS11(Read := "Unit1.CM_Name".ReadFromHMI,   // "LER_CM_Name"
               Write := "Unit1.CM_Name".WriteToHMI,
               StartArr := 11,
               CntAr := 2,
               HMIAxis_1 := "Unit1.Em4.HmiInterface".cmAnodeMainPnP1AxisY.configuration.referenceDesignator,
               HMIAxis_2 := "Unit1.Em4.HmiInterface".cmAnodeMainPnP1AxisZ.configuration.referenceDesignator,
               HMIAxis_3 := #AXIS11.Temp,
               HMIAxis_4 := #AXIS11.Temp,
               HMIAxis_5 := #AXIS11.Temp,
               Config_1 := "Unit1.Em4.Config".cmAnodeMainPnP1AxisY.referenceDesignator,
               Config_2 := "Unit1.Em4.Config".cmAnodeMainPnP1AxisZ.referenceDesignator,
               Config_3 := #AXIS11.Temp,
               Config_4 := #AXIS11.Temp,
               Config_5 := #AXIS11.Temp,
               NameManDB := "Unit1.CM_Name".AxisName);
   END_IF;
   #AXIS14(Read := "Unit1.CM_Name".ReadFromHMI,   // "LER_CM_Name"
           Write := "Unit1.CM_Name".WriteToHMI,
           StartArr := 14,
           CntAr := 4,
           HMIAxis_1 := "Unit1.Em4.HmiInterface".cmAnodeMainPnP2AxisZ.configuration.referenceDesignator,
           HMIAxis_2 := "Unit1.Em4.HmiInterface".cmAnodeAlignTableAxisX.configuration.referenceDesignator,
           HMIAxis_3 := "Unit1.Em4.HmiInterface".cmAnodeAlignTableAxisY1.configuration.referenceDesignator,
           HMIAxis_4 := "Unit1.Em4.HmiInterface".cmAnodeAlignTableAxisY2.configuration.referenceDesignator,
           HMIAxis_5 := #AXIS14.Temp,
           Config_1 := "Unit1.Em4.Config".cmAnodeMainPnP2AxisZ.referenceDesignator,
           Config_2 := "Unit1.Em4.Config".cmAnodeAlignTableAxisX.referenceDesignator,
           Config_3 := "Unit1.Em4.Config".cmAnodeAlignTableAxisY1.referenceDesignator,
           Config_4 := "Unit1.Em4.Config".cmAnodeAlignTableAxisY2.referenceDesignator,
           Config_5 := #AXIS14.Temp,
           NameManDB := "Unit1.CM_Name".AxisName);
END_REGION

REGION Network 314: Cylinder
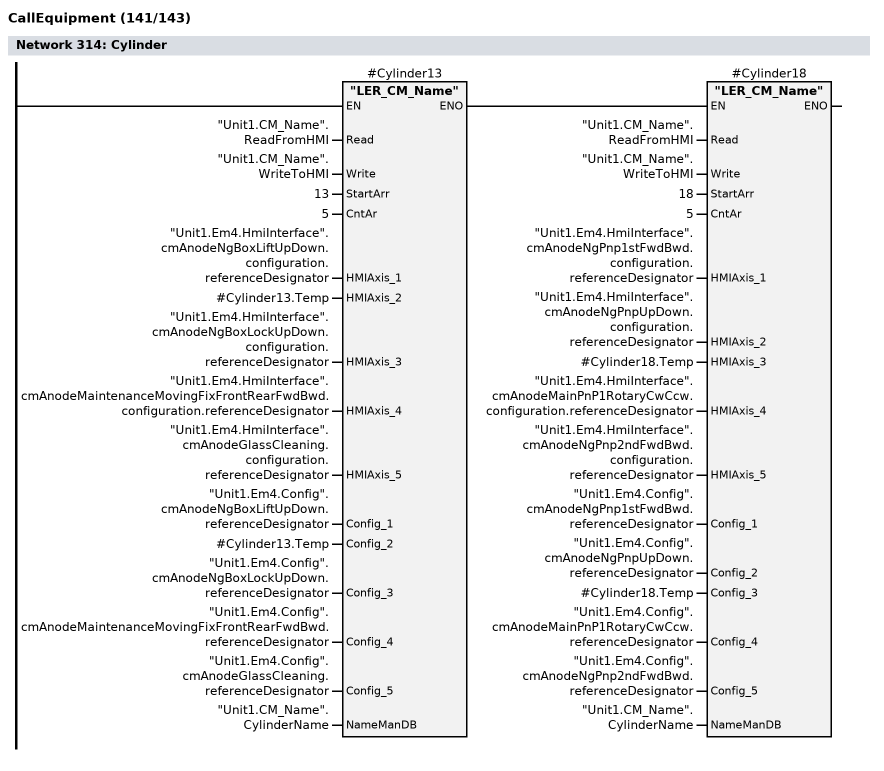
   RUNG wire#powerrail
      #Cylinder13(Read := "Unit1.CM_Name".ReadFromHMI, Write := "Unit1.CM_Name".WriteToHMI, StartArr := 13, CntAr := 5, HMIAxis_1 := "Unit1.Em4.HmiInterface".cmAnodeNgBoxLiftUpDown.configuration.referenceDesignator, HMIAxis_2 := #Cylinder13.Temp, HMIAxis_3 := "Unit1.Em4.HmiInterface".cmAnodeNgBoxLockUpDown.configuration.referenceDesignator, HMIAxis_4 := "Unit1.Em4.HmiInterface".cmAnodeMaintenanceMovingFixFrontRearFwdBwd.configuration.referenceDesignator, HMIAxis_5 := "Unit1.Em4.HmiInterface".cmAnodeGlassCleaning.configuration.referenceDesignator, Config_1 := "Unit1.Em4.Config".cmAnodeNgBoxLiftUpDown.referenceDesignator, Config_2 := #Cylinder13.Temp, Config_3 := "Unit1.Em4.Config".cmAnodeNgBoxLockUpDown.referenceDesignator, Config_4 := "Unit1.Em4.Config".cmAnodeMaintenanceMovingFixFrontRearFwdBwd.referenceDesignator, Config_5 := "Unit1.Em4.Config".cmAnodeGlassCleaning.referenceDesignator, NameManDB := "Unit1.CM_Name".CylinderName)
      #Cylinder18(Read := "Unit1.CM_Name".ReadFromHMI, Write := "Unit1.CM_Name".WriteToHMI, StartArr := 18, CntAr := 5, HMIAxis_1 := "Unit1.Em4.HmiInterface".cmAnodeNgPnp1stFwdBwd.configuration.referenceDesignator, HMIAxis_2 := "Unit1.Em4.HmiInterface".cmAnodeNgPnpUpDown.configuration.referenceDesignator, HMIAxis_3 := #Cylinder18.Temp, HMIAxis_4 := "Unit1.Em4.HmiInterface".cmAnodeMainPnP1RotaryCwCcw.configuration.referenceDesignator, HMIAxis_5 := "Unit1.Em4.HmiInterface".cmAnodeNgPnp2ndFwdBwd.configuration.referenceDesignator, Config_1 := "Unit1.Em4.Config".cmAnodeNgPnp1stFwdBwd.referenceDesignator, Config_2 := "Unit1.Em4.Config".cmAnodeNgPnpUpDown.referenceDesignator, Config_3 := #Cylinder18.Temp, Config_4 := "Unit1.Em4.Config".cmAnodeMainPnP1RotaryCwCcw.referenceDesignator, Config_5 := "Unit1.Em4.Config".cmAnodeNgPnp2ndFwdBwd.referenceDesignator, NameManDB := "Unit1.CM_Name".CylinderName)
   END_RUNG
   // the same network as SCL:
   #Cylinder13(Read := "Unit1.CM_Name".ReadFromHMI,   // "LER_CM_Name"
               Write := "Unit1.CM_Name".WriteToHMI,
               StartArr := 13,
               CntAr := 5,
               HMIAxis_1 := "Unit1.Em4.HmiInterface".cmAnodeNgBoxLiftUpDown.configuration.referenceDesignator,
               HMIAxis_2 := #Cylinder13.Temp,
               HMIAxis_3 := "Unit1.Em4.HmiInterface".cmAnodeNgBoxLockUpDown.configuration.referenceDesignator,
               HMIAxis_4 := "Unit1.Em4.HmiInterface".cmAnodeMaintenanceMovingFixFrontRearFwdBwd.configuration.referenceDesignator,
               HMIAxis_5 := "Unit1.Em4.HmiInterface".cmAnodeGlassCleaning.configuration.referenceDesignator,
               Config_1 := "Unit1.Em4.Config".cmAnodeNgBoxLiftUpDown.referenceDesignator,
               Config_2 := #Cylinder13.Temp,
               Config_3 := "Unit1.Em4.Config".cmAnodeNgBoxLockUpDown.referenceDesignator,
               Config_4 := "Unit1.Em4.Config".cmAnodeMaintenanceMovingFixFrontRearFwdBwd.referenceDesignator,
               Config_5 := "Unit1.Em4.Config".cmAnodeGlassCleaning.referenceDesignator,
               NameManDB := "Unit1.CM_Name".CylinderName,
               ENO => #_w1);
   IF #_w1 THEN
       #Cylinder18(Read := "Unit1.CM_Name".ReadFromHMI,   // "LER_CM_Name"
                   Write := "Unit1.CM_Name".WriteToHMI,
                   StartArr := 18,
                   CntAr := 5,
                   HMIAxis_1 := "Unit1.Em4.HmiInterface".cmAnodeNgPnp1stFwdBwd.configuration.referenceDesignator,
                   HMIAxis_2 := "Unit1.Em4.HmiInterface".cmAnodeNgPnpUpDown.configuration.referenceDesignator,
                   HMIAxis_3 := #Cylinder18.Temp,
                   HMIAxis_4 := "Unit1.Em4.HmiInterface".cmAnodeMainPnP1RotaryCwCcw.configuration.referenceDesignator,
                   HMIAxis_5 := "Unit1.Em4.HmiInterface".cmAnodeNgPnp2ndFwdBwd.configuration.referenceDesignator,
                   Config_1 := "Unit1.Em4.Config".cmAnodeNgPnp1stFwdBwd.referenceDesignator,
                   Config_2 := "Unit1.Em4.Config".cmAnodeNgPnpUpDown.referenceDesignator,
                   Config_3 := #Cylinder18.Temp,
                   Config_4 := "Unit1.Em4.Config".cmAnodeMainPnP1RotaryCwCcw.referenceDesignator,
                   Config_5 := "Unit1.Em4.Config".cmAnodeNgPnp2ndFwdBwd.referenceDesignator,
                   NameManDB := "Unit1.CM_Name".CylinderName);
   END_IF;
END_REGION

REGION Network 315: Vaccum
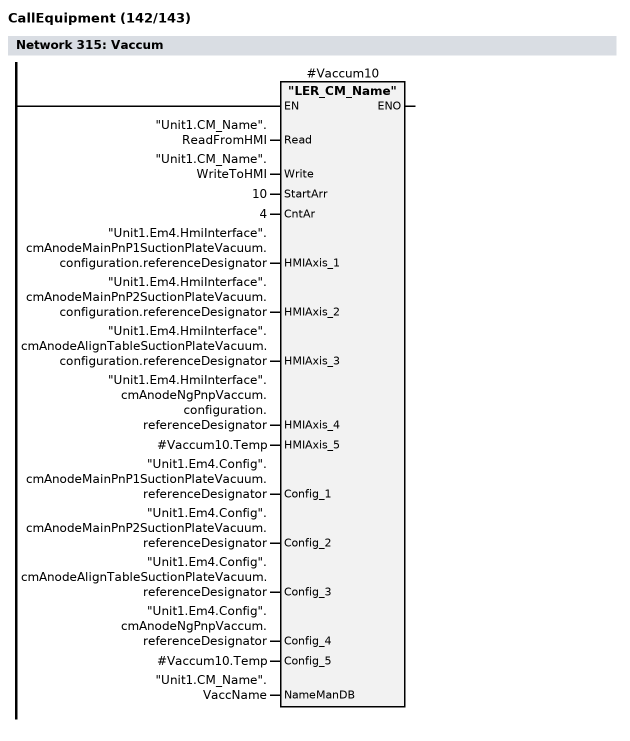
   RUNG wire#powerrail
      #Vaccum10(Read := "Unit1.CM_Name".ReadFromHMI, Write := "Unit1.CM_Name".WriteToHMI, StartArr := 10, CntAr := 4, HMIAxis_1 := "Unit1.Em4.HmiInterface".cmAnodeMainPnP1SuctionPlateVacuum.configuration.referenceDesignator, HMIAxis_2 := "Unit1.Em4.HmiInterface".cmAnodeMainPnP2SuctionPlateVacuum.configuration.referenceDesignator, HMIAxis_3 := "Unit1.Em4.HmiInterface".cmAnodeAlignTableSuctionPlateVacuum.configuration.referenceDesignator, HMIAxis_4 := "Unit1.Em4.HmiInterface".cmAnodeNgPnpVaccum.configuration.referenceDesignator, HMIAxis_5 := #Vaccum10.Temp, Config_1 := "Unit1.Em4.Config".cmAnodeMainPnP1SuctionPlateVacuum.referenceDesignator, Config_2 := "Unit1.Em4.Config".cmAnodeMainPnP2SuctionPlateVacuum.referenceDesignator, Config_3 := "Unit1.Em4.Config".cmAnodeAlignTableSuctionPlateVacuum.referenceDesignator, Config_4 := "Unit1.Em4.Config".cmAnodeNgPnpVaccum.referenceDesignator, Config_5 := #Vaccum10.Temp, NameManDB := "Unit1.CM_Name".VaccName)
   END_RUNG
   // the same network as SCL:
   #Vaccum10(Read := "Unit1.CM_Name".ReadFromHMI,   // "LER_CM_Name"
             Write := "Unit1.CM_Name".WriteToHMI,
             StartArr := 10,
             CntAr := 4,
             HMIAxis_1 := "Unit1.Em4.HmiInterface".cmAnodeMainPnP1SuctionPlateVacuum.configuration.referenceDesignator,
             HMIAxis_2 := "Unit1.Em4.HmiInterface".cmAnodeMainPnP2SuctionPlateVacuum.configuration.referenceDesignator,
             HMIAxis_3 := "Unit1.Em4.HmiInterface".cmAnodeAlignTableSuctionPlateVacuum.configuration.referenceDesignator,
             HMIAxis_4 := "Unit1.Em4.HmiInterface".cmAnodeNgPnpVaccum.configuration.referenceDesignator,
             HMIAxis_5 := #Vaccum10.Temp,
             Config_1 := "Unit1.Em4.Config".cmAnodeMainPnP1SuctionPlateVacuum.referenceDesignator,
             Config_2 := "Unit1.Em4.Config".cmAnodeMainPnP2SuctionPlateVacuum.referenceDesignator,
             Config_3 := "Unit1.Em4.Config".cmAnodeAlignTableSuctionPlateVacuum.referenceDesignator,
             Config_4 := "Unit1.Em4.Config".cmAnodeNgPnpVaccum.referenceDesignator,
             Config_5 := #Vaccum10.Temp,
             NameManDB := "Unit1.CM_Name".VaccName);
END_REGION

REGION Network 316: BA015 Interface Data
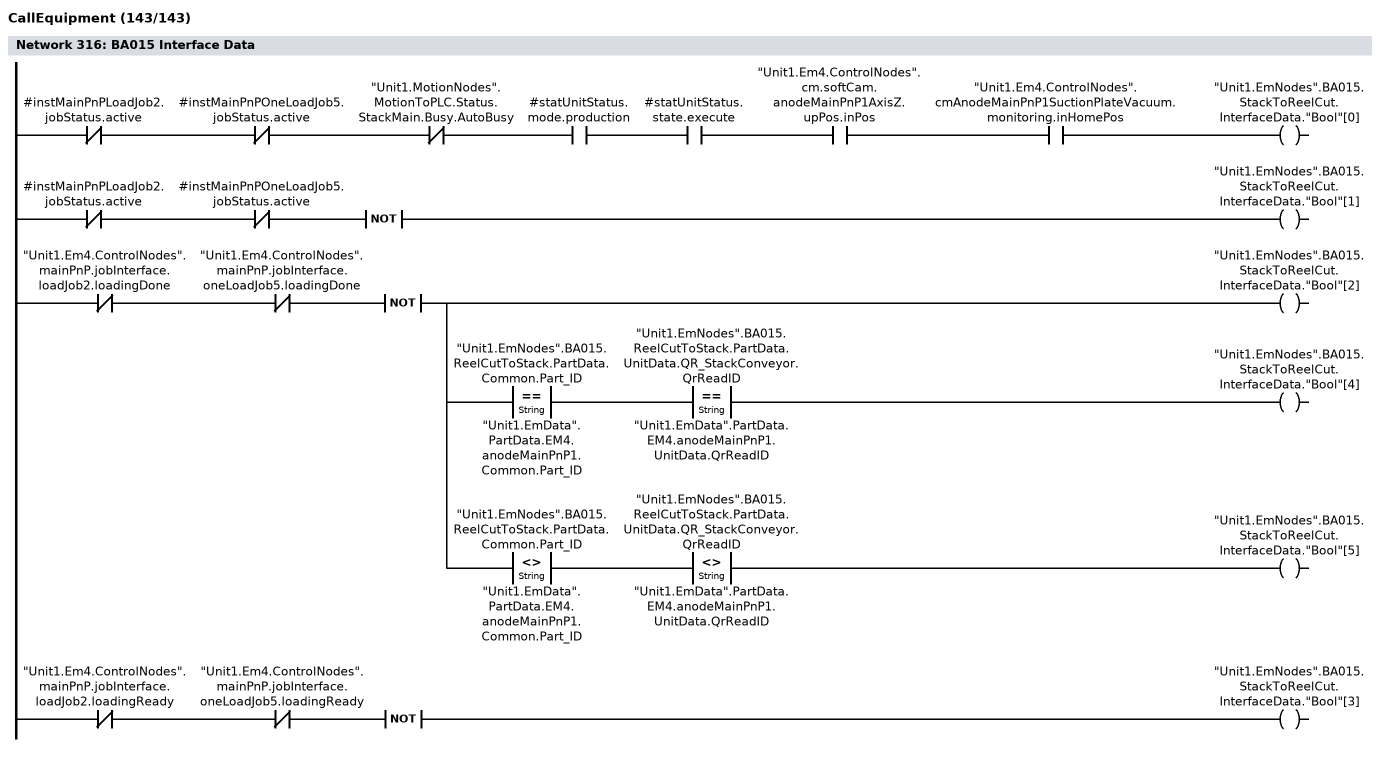
   RUNG wire#powerrail
      I_Contact( #instMainPnPLoadJob2.jobStatus.active )
      I_Contact( #instMainPnPOneLoadJob5.jobStatus.active )
      I_Contact( "Unit1.MotionNodes".MotionToPLC.Status.StackMain.Busy.AutoBusy )
      Contact( #statUnitStatus.mode.production )
      Contact( #statUnitStatus.state.execute )
      Contact( "Unit1.Em4.ControlNodes".cm.softCam.anodeMainPnP1AxisZ.upPos.inPos )
      Contact( "Unit1.Em4.ControlNodes".cmAnodeMainPnP1SuctionPlateVacuum.monitoring.inHomePos )
      Coil( "Unit1.EmNodes".BA015.StackToReelCut.InterfaceData."Bool"[0] )
   END_RUNG
   RUNG wire#powerrail
      I_Contact( #instMainPnPLoadJob2.jobStatus.active )
      I_Contact( #instMainPnPOneLoadJob5.jobStatus.active )
      Not()
      Coil( "Unit1.EmNodes".BA015.StackToReelCut.InterfaceData."Bool"[1] )
   END_RUNG
   RUNG wire#powerrail
      I_Contact( "Unit1.Em4.ControlNodes".mainPnP.jobInterface.loadJob2.loadingDone )
      I_Contact( "Unit1.Em4.ControlNodes".mainPnP.jobInterface.oneLoadJob5.loadingDone )
      Not()
      wire#w1
      Coil( "Unit1.EmNodes".BA015.StackToReelCut.InterfaceData."Bool"[2] )
   END_RUNG
   RUNG wire#w1
      { S7_Templates := "SrcType := String" } EQ_Contact(in1 := "Unit1.EmNodes".BA015.ReelCutToStack.PartData.Common.Part_ID, in2 := "Unit1.EmData".PartData.EM4.anodeMainPnP1.Common.Part_ID)
      { S7_Templates := "SrcType := String" } EQ_Contact(in1 := "Unit1.EmNodes".BA015.ReelCutToStack.PartData.UnitData.QR_StackConveyor.QrReadID, in2 := "Unit1.EmData".PartData.EM4.anodeMainPnP1.UnitData.QrReadID)
      Coil( "Unit1.EmNodes".BA015.StackToReelCut.InterfaceData."Bool"[4] )
   END_RUNG
   RUNG wire#w1
      { S7_Templates := "SrcType := String" } NE_Contact(in1 := "Unit1.EmNodes".BA015.ReelCutToStack.PartData.Common.Part_ID, in2 := "Unit1.EmData".PartData.EM4.anodeMainPnP1.Common.Part_ID)
      { S7_Templates := "SrcType := String" } NE_Contact(in1 := "Unit1.EmNodes".BA015.ReelCutToStack.PartData.UnitData.QR_StackConveyor.QrReadID, in2 := "Unit1.EmData".PartData.EM4.anodeMainPnP1.UnitData.QrReadID)
      Coil( "Unit1.EmNodes".BA015.StackToReelCut.InterfaceData."Bool"[5] )
   END_RUNG
   RUNG wire#powerrail
      I_Contact( "Unit1.Em4.ControlNodes".mainPnP.jobInterface.loadJob2.loadingReady )
      I_Contact( "Unit1.Em4.ControlNodes".mainPnP.jobInterface.oneLoadJob5.loadingReady )
      Not()
      Coil( "Unit1.EmNodes".BA015.StackToReelCut.InterfaceData."Bool"[3] )
   END_RUNG
   // the same network as SCL:
   "Unit1.EmNodes".BA015.StackToReelCut.InterfaceData."Bool"[0] := NOT #instMainPnPLoadJob2.jobStatus.active AND NOT #instMainPnPOneLoadJob5.jobStatus.active AND NOT "Unit1.MotionNodes".MotionToPLC.Status.StackMain.Busy.AutoBusy AND #statUnitStatus.mode.production AND #statUnitStatus.state.execute AND "Unit1.Em4.ControlNodes".cm.softCam.anodeMainPnP1AxisZ.upPos.inPos AND "Unit1.Em4.ControlNodes".cmAnodeMainPnP1SuctionPlateVacuum.monitoring.inHomePos;
   "Unit1.EmNodes".BA015.StackToReelCut.InterfaceData."Bool"[1] := NOT (NOT #instMainPnPLoadJob2.jobStatus.active AND NOT #instMainPnPOneLoadJob5.jobStatus.active);
   "Unit1.EmNodes".BA015.StackToReelCut.InterfaceData."Bool"[2] := NOT (NOT "Unit1.Em4.ControlNodes".mainPnP.jobInterface.loadJob2.loadingDone AND NOT "Unit1.Em4.ControlNodes".mainPnP.jobInterface.oneLoadJob5.loadingDone);
   "Unit1.EmNodes".BA015.StackToReelCut.InterfaceData."Bool"[4] := NOT (NOT "Unit1.Em4.ControlNodes".mainPnP.jobInterface.loadJob2.loadingDone AND NOT "Unit1.Em4.ControlNodes".mainPnP.jobInterface.oneLoadJob5.loadingDone) AND ("Unit1.EmNodes".BA015.ReelCutToStack.PartData.Common.Part_ID = "Unit1.EmData".PartData.EM4.anodeMainPnP1.Common.Part_ID) AND ("Unit1.EmNodes".BA015.ReelCutToStack.PartData.UnitData.QR_StackConveyor.QrReadID = "Unit1.EmData".PartData.EM4.anodeMainPnP1.UnitData.QrReadID);
   "Unit1.EmNodes".BA015.StackToReelCut.InterfaceData."Bool"[5] := NOT (NOT "Unit1.Em4.ControlNodes".mainPnP.jobInterface.loadJob2.loadingDone AND NOT "Unit1.Em4.ControlNodes".mainPnP.jobInterface.oneLoadJob5.loadingDone) AND ("Unit1.EmNodes".BA015.ReelCutToStack.PartData.Common.Part_ID <> "Unit1.EmData".PartData.EM4.anodeMainPnP1.Common.Part_ID) AND ("Unit1.EmNodes".BA015.ReelCutToStack.PartData.UnitData.QR_StackConveyor.QrReadID <> "Unit1.EmData".PartData.EM4.anodeMainPnP1.UnitData.QrReadID);
   "Unit1.EmNodes".BA015.StackToReelCut.InterfaceData."Bool"[3] := NOT (NOT "Unit1.Em4.ControlNodes".mainPnP.jobInterface.loadJob2.loadingReady AND NOT "Unit1.Em4.ControlNodes".mainPnP.jobInterface.oneLoadJob5.loadingReady);
END_REGION
END_FUNCTION_BLOCK
